LIN {X 0,Y 445.555,Z 224.747,A -85,B 0,C 180,E1 -8713.867,E2 -8713.867} C_VEL
LIN {X 0,Y 447.569,Z 235.644,A -85,B 0,C 180,E1 -8714.246,E2 -8714.246} C_VEL
LIN {X 0,Y 449.181,Z 245.497,A -85,B 0,C 180,E1 -8714.691,E2 -8714.691} C_VEL
LIN {X 0,Y 449.133,Z 253.576,A -85,B 0,C 180,E1 -8715.096,E2 -8715.096} C_VEL
LIN {X 0,Y 448.605,Z 263.719,A -85,B 0,C 180,E1 -8715.715,E2 -8715.715} C_VEL
LIN {X 0,Y 448.134,Z 272.72,A -85,B 0,C 180,E1 -8716.394,E2 -8716.394} C_VEL
LIN {X 0,Y 447.699,Z 281.135,A -85,B 0,C 180,E1 -8717.157,E2 -8717.157} C_VEL
LIN {X 0,Y 447.283,Z 288.853,A -85,B 0,C 180,E1 -8717.984,E2 -8717.984} C_VEL
LIN {X 0,Y 446.817,Z 296.075,A -85,B 0,C 180,E1 -8718.891,E2 -8718.891} C_VEL
LIN {X 0,Y 446.49,Z 302.281,A -85,B 0,C 180,E1 -8719.8,E2 -8719.8} C_VEL
LIN {X 0,Y 446.129,Z 308.821,A -85,B 0,C 180,E1 -8720.936,E2 -8720.936} C_VEL
LIN {X 0,Y 445.886,Z 313.324,A -85,B 0,C 180,E1 -8721.845,E2 -8721.845} C_VEL
LIN {X 0,Y 445.655,Z 318.973,A -85,B 0,C 180,E1 -8723.253,E2 -8723.253} C_VEL
LIN {X 0,Y 445.538,Z 323.142,A -85,B 0,C 180,E1 -8724.569,E2 -8724.569} C_VEL
LIN {X 0,Y 445.43,Z 325.507,A -85,B 0,C 180,E1 -8725.475,E2 -8725.475} C_VEL
LIN {X 0,Y 445.391,Z 327.304,A -85,B 0,C 180,E1 -8726.381,E2 -8726.381} C_VEL
LIN {X 0,Y 445.353,Z 329.747,A -85,B 0,C 180,E1 -8728.191,E2 -8728.191} C_VEL
LIN {X 0,Y 445.315,Z 330.334,A -85,B 0,C 180,E1 -8729.096,E2 -8729.096} C_VEL
LIN {X 0,Y 445.315,Z 330.334,A -85,B 0,C 180,E1 -8730.904,E2 -8730.904} C_VEL
LIN {X 0,Y 445.353,Z 329.747,A -85,B 0,C 180,E1 -8731.809,E2 -8731.809} C_VEL
LIN {X 0,Y 445.391,Z 327.304,A -85,B 0,C 180,E1 -8733.619,E2 -8733.619} C_VEL
LIN {X 0,Y 445.5,Z 324.359,A -85,B 0,C 180,E1 -8734.977,E2 -8734.977} C_VEL
LIN {X 0,Y 445.579,Z 320.37,A -85,B 0,C 180,E1 -8736.339,E2 -8736.339} C_VEL
LIN {X 0,Y 445.762,Z 315.239,A -85,B 0,C 180,E1 -8737.701,E2 -8737.701} C_VEL
LIN {X 0,Y 446.078,Z 309.978,A -85,B 0,C 180,E1 -8738.836,E2 -8738.836} C_VEL
LIN {X 0,Y 446.426,Z 303.658,A -85,B 0,C 180,E1 -8739.972,E2 -8739.972} C_VEL
LIN {X 0,Y 446.703,Z 297.702,A -85,B 0,C 180,E1 -8740.882,E2 -8740.882} C_VEL
LIN {X 0,Y 447.153,Z 290.773,A -85,B 0,C 180,E1 -8741.79,E2 -8741.79} C_VEL
LIN {X 0,Y 447.622,Z 282.589,A -85,B 0,C 180,E1 -8742.698,E2 -8742.698} C_VEL
LIN {X 0,Y 448.019,Z 274.012,A -85,B 0,C 180,E1 -8743.499,E2 -8743.499} C_VEL
LIN {X 0,Y 448.505,Z 265.351,A -85,B 0,C 180,E1 -8744.172,E2 -8744.172} C_VEL
LIN {X 0,Y 448.992,Z 255.589,A -85,B 0,C 180,E1 -8744.793,E2 -8744.793} C_VEL
LIN {X 0,Y 449.335,Z 246.791,A -85,B 0,C 180,E1 -8745.246,E2 -8745.246} C_VEL
LIN {X 0,Y 447.725,Z 236.462,A -85,B 0,C 180,E1 -8745.721,E2 -8745.721} C_VEL
LIN {X 0,Y 445.687,Z 225.777,A -85,B 0,C 180,E1 -8746.102,E2 -8746.102} C_VEL
LIN {X 0,Y 445.555,Z 224.693,A -85,B 0,C 180,E1 -8746.161,E2 -8746.161} C_VEL
LIN {X 0,Y 445.687,Z 218.655,A -85,B 0,C 180,E1 -8749.338,E2 -8749.338} C_VEL
LIN {X 0,Y 445.855,Z 213.313,A -85,B 0,C 180,E1 -8752.229,E2 -8752.229} C_VEL
LIN {X 0,Y 446.032,Z 208.032,A -85,B 0,C 180,E1 -8755.178,E2 -8755.178} C_VEL
LIN {X 0,Y 446.268,Z 202.816,A -85,B 0,C 180,E1 -8758.193,E2 -8758.193} C_VEL
LIN {X 0,Y 446.557,Z 196.849,A -85,B 0,C 180,E1 -8761.803,E2 -8761.803} C_VEL
LIN {X 0,Y 446.894,Z 191.658,A -85,B 0,C 180,E1 -8765.137,E2 -8765.137} C_VEL
LIN {X 0,Y 447.241,Z 187.135,A -85,B 0,C 180,E1 -8768.213,E2 -8768.213} C_VEL
LIN {X 0,Y 447.459,Z 182.971,A -85,B 0,C 180,E1 -8771.274,E2 -8771.274} C_VEL
LIN {X 0,Y 447.256,Z 179.884,A -85,B 0,C 180,E1 -8773.74,E2 -8773.74} C_VEL
LIN {X 0,Y 446.776,Z 176.867,A -85,B 0,C 180,E1 -8776.352,E2 -8776.352} C_VEL
LIN {X 0,Y 446.43,Z 174.429,A -85,B 0,C 180,E1 -8778.609,E2 -8778.609} C_VEL
LIN {X 0,Y 446.438,Z 174.378,A -85,B 0,C 180,E1 -8780.972,E2 -8780.972} C_VEL
LIN {X 0,Y 446.416,Z 174.377,A -85,B 0,C 180,E1 -8784.373,E2 -8784.373} C_VEL
LIN {X 0,Y 446.419,Z 174.373,A -85,B 0,C 180,E1 -8787.638,E2 -8787.638} C_VEL
LIN {X 0,Y 446.444,Z 174.374,A -85,B 0,C 180,E1 -8790.79,E2 -8790.79} C_VEL
LIN {X 0,Y 446.474,Z 174.367,A -85,B 0,C 180,E1 -8793.848,E2 -8793.848} C_VEL
LIN {X 0,Y 446.425,Z 174.375,A -85,B 0,C 180,E1 -8796.823,E2 -8796.823} C_VEL
LIN {X 0,Y 446.44,Z 174.372,A -85,B 0,C 180,E1 -8799.736,E2 -8799.736} C_VEL
LIN {X 0,Y 446.458,Z 174.371,A -85,B 0,C 180,E1 -8802.596,E2 -8802.596} C_VEL
LIN {X 0,Y 446.465,Z 174.368,A -85,B 0,C 180,E1 -8805.412,E2 -8805.412} C_VEL
LIN {X 0,Y 446.512,Z 174.367,A -85,B 0,C 180,E1 -8808.192,E2 -8808.192} C_VEL
LIN {X 0,Y 446.595,Z 174.358,A -85,B 0,C 180,E1 -8811.857,E2 -8811.857} C_VEL
LIN {X 0,Y 446.637,Z 174.346,A -85,B 0,C 180,E1 -8814.582,E2 -8814.582} C_VEL
LIN {X 0,Y 446.657,Z 174.346,A -85,B 0,C 180,E1 -8818.196,E2 -8818.196} C_VEL
LIN {X 0,Y 446.787,Z 174.331,A -85,B 0,C 180,E1 -8820,E2 -8820} C_VEL
LIN {X 0,Y 446.685,Z 174.34,A -85,B 0,C 180,E1 -8822.705,E2 -8822.705} C_VEL
LIN {X 0,Y 446.64,Z 174.346,A -85,B 0,C 180,E1 -8826.323,E2 -8826.323} C_VEL
LIN {X 0,Y 446.532,Z 174.362,A -85,B 0,C 180,E1 -8829.055,E2 -8829.055} C_VEL
LIN {X 0,Y 446.515,Z 174.362,A -85,B 0,C 180,E1 -8832.729,E2 -8832.729} C_VEL
LIN {X 0,Y 446.49,Z 174.364,A -85,B 0,C 180,E1 -8836.228,E2 -8836.228} C_VEL
LIN {X 0,Y 446.463,Z 174.373,A -85,B 0,C 180,E1 -8839.303,E2 -8839.303} C_VEL
LIN {X 0,Y 446.411,Z 174.374,A -85,B 0,C 180,E1 -8842.199,E2 -8842.199} C_VEL
LIN {X 0,Y 446.451,Z 174.374,A -85,B 0,C 180,E1 -8845.152,E2 -8845.152} C_VEL
LIN {X 0,Y 446.478,Z 174.366,A -85,B 0,C 180,E1 -8848.178,E2 -8848.178} C_VEL
LIN {X 0,Y 446.413,Z 174.375,A -85,B 0,C 180,E1 -8851.3,E2 -8851.3} C_VEL
LIN {X 0,Y 446.424,Z 174.378,A -85,B 0,C 180,E1 -8854.523,E2 -8854.523} C_VEL
LIN {X 0,Y 446.43,Z 174.374,A -85,B 0,C 180,E1 -8858.083,E2 -8858.083} C_VEL
LIN {X 0,Y 446.437,Z 174.373,A -85,B 0,C 180,E1 -8860.92,E2 -8860.92} C_VEL
LIN {X 0,Y 446.395,Z 174.378,A -85,B 0,C 180,E1 -8863.846,E2 -8863.846} C_VEL
LIN {X 0,Y 446.409,Z 174.381,A -85,B 0,C 180,E1 -8866.401,E2 -8866.401} C_VEL
LIN {X 0,Y 446.445,Z 174.373,A -85,B 0,C 180,E1 -8869.803,E2 -8869.803} C_VEL
LIN {X 0,Y 446.422,Z 174.38,A -85,B 0,C 180,E1 -8872.123,E2 -8872.123} C_VEL
LIN {X 0,Y 446.425,Z 174.374,A -85,B 0,C 180,E1 -8875.477,E2 -8875.477} C_VEL
LIN {X 0,Y 446.415,Z 174.374,A -85,B 0,C 180,E1 -8878.7,E2 -8878.7} C_VEL
LIN {X 0,Y 446.48,Z 174.373,A -85,B 0,C 180,E1 -8881.821,E2 -8881.821} C_VEL
LIN {X 0,Y 446.453,Z 174.369,A -85,B 0,C 180,E1 -8884.848,E2 -8884.848} C_VEL
LIN {X 0,Y 446.444,Z 174.371,A -85,B 0,C 180,E1 -8888.245,E2 -8888.245} C_VEL
LIN {X 0,Y 446.454,Z 174.376,A -85,B 0,C 180,E1 -8891.649,E2 -8891.649} C_VEL
LIN {X 0,Y 446.505,Z 174.366,A -85,B 0,C 180,E1 -8894.48,E2 -8894.48} C_VEL
LIN {X 0,Y 446.514,Z 174.364,A -85,B 0,C 180,E1 -8898.193,E2 -8898.193} C_VEL
LIN {X 0,Y 446.597,Z 174.355,A -85,B 0,C 180,E1 -8901.858,E2 -8901.858} C_VEL
LIN {X 0,Y 446.644,Z 174.349,A -85,B 0,C 180,E1 -8904.583,E2 -8904.583} C_VEL
LIN {X 0,Y 446.619,Z 174.353,A -85,B 0,C 180,E1 -8907.001,E2 -8907.001} C_VEL
LIN {X 0,Y 446.101,Z 174.421,A -85,B 0,C 180,E1 -8907.754,E2 -8907.754} C_VEL
LIN {X 0,Y 443.286,Z 174.777,A -85,B 0,C 180,E1 -8908.977,E2 -8908.977} C_VEL
LIN {X 0,Y 440.802,Z 175.085,A -85,B 0,C 180,E1 -8909.964,E2 -8909.964} C_VEL
LIN {X 0,Y 439.713,Z 175.216,A -85,B 0,C 180,E1 -8910.727,E2 -8910.727} C_VEL
LIN {X 0,Y 439.619,Z 175.225,A -85,B 0,C 180,E1 -8910.986,E2 -8910.986} C_VEL
LIN {X 0,Y 439.653,Z 175.222,A -85,B 0,C 180,E1 -8912.749,E2 -8912.749} C_VEL
LIN {X 0,Y 439.616,Z 175.227,A -85,B 0,C 180,E1 -8916.425,E2 -8916.425} C_VEL
LIN {X 0,Y 439.497,Z 175.24,A -85,B 0,C 180,E1 -8919.202,E2 -8919.202} C_VEL
LIN {X 0,Y 439.462,Z 175.246,A -85,B 0,C 180,E1 -8922.938,E2 -8922.938} C_VEL
LIN {X 0,Y 439.443,Z 175.248,A -85,B 0,C 180,E1 -8926.349,E2 -8926.349} C_VEL
LIN {X 0,Y 439.399,Z 175.248,A -85,B 0,C 180,E1 -8929.626,E2 -8929.626} C_VEL
LIN {X 0,Y 439.362,Z 175.256,A -85,B 0,C 180,E1 -8932.575,E2 -8932.575} C_VEL
LIN {X 0,Y 439.4,Z 175.248,A -85,B 0,C 180,E1 -8935.585,E2 -8935.585} C_VEL
LIN {X 0,Y 439.42,Z 175.246,A -85,B 0,C 180,E1 -8938.673,E2 -8938.673} C_VEL
LIN {X 0,Y 439.378,Z 175.258,A -85,B 0,C 180,E1 -8942.033,E2 -8942.033} C_VEL
LIN {X 0,Y 439.391,Z 175.25,A -85,B 0,C 180,E1 -8945.341,E2 -8945.341} C_VEL
LIN {X 0,Y 439.39,Z 175.249,A -85,B 0,C 180,E1 -8948.594,E2 -8948.594} C_VEL
LIN {X 0,Y 439.392,Z 175.25,A -85,B 0,C 180,E1 -8951.258,E2 -8951.258} C_VEL
LIN {X 0,Y 439.395,Z 175.248,A -85,B 0,C 180,E1 -8954.729,E2 -8954.729} C_VEL
LIN {X 0,Y 439.391,Z 175.253,A -85,B 0,C 180,E1 -8957.796,E2 -8957.796} C_VEL
LIN {X 0,Y 439.444,Z 175.242,A -85,B 0,C 180,E1 -8960.23,E2 -8960.23} C_VEL
LIN {X 0,Y 439.371,Z 175.255,A -85,B 0,C 180,E1 -8963.713,E2 -8963.713} C_VEL
LIN {X 0,Y 439.366,Z 175.256,A -85,B 0,C 180,E1 -8967.054,E2 -8967.054} C_VEL
LIN {X 0,Y 439.39,Z 175.249,A -85,B 0,C 180,E1 -8970.275,E2 -8970.275} C_VEL
LIN {X 0,Y 439.427,Z 175.246,A -85,B 0,C 180,E1 -8973.589,E2 -8973.589} C_VEL
LIN {X 0,Y 439.38,Z 175.251,A -85,B 0,C 180,E1 -8976.43,E2 -8976.43} C_VEL
LIN {X 0,Y 439.382,Z 175.252,A -85,B 0,C 180,E1 -8979.397,E2 -8979.397} C_VEL
LIN {X 0,Y 439.425,Z 175.246,A -85,B 0,C 180,E1 -8982.31,E2 -8982.31} C_VEL
LIN {X 0,Y 439.442,Z 175.245,A -85,B 0,C 180,E1 -8985.174,E2 -8985.174} C_VEL
LIN {X 0,Y 439.477,Z 175.239,A -85,B 0,C 180,E1 -8988.002,E2 -8988.002} C_VEL
LIN {X 0,Y 439.542,Z 175.23,A -85,B 0,C 180,E1 -8991.727,E2 -8991.727} C_VEL
LIN {X 0,Y 439.614,Z 175.228,A -85,B 0,C 180,E1 -8994.496,E2 -8994.496} C_VEL
LIN {X 0,Y 439.628,Z 175.224,A -85,B 0,C 180,E1 -8998.168,E2 -8998.168} C_VEL
LIN {X 0,Y 439.757,Z 175.206,A -85,B 0,C 180,E1 -9000,E2 -9000} C_VEL
LIN {X 0,Y 439.634,Z 175.22,A -85,B 0,C 180,E1 -9002.749,E2 -9002.749} C_VEL
LIN {X 0,Y 439.607,Z 175.225,A -85,B 0,C 180,E1 -9006.426,E2 -9006.426} C_VEL
LIN {X 0,Y 439.495,Z 175.236,A -85,B 0,C 180,E1 -9009.202,E2 -9009.202} C_VEL
LIN {X 0,Y 439.461,Z 175.24,A -85,B 0,C 180,E1 -9012.938,E2 -9012.938} C_VEL
LIN {X 0,Y 439.443,Z 175.244,A -85,B 0,C 180,E1 -9016.349,E2 -9016.349} C_VEL
LIN {X 0,Y 439.398,Z 175.254,A -85,B 0,C 180,E1 -9019.627,E2 -9019.627} C_VEL
LIN {X 0,Y 439.361,Z 175.252,A -85,B 0,C 180,E1 -9022.576,E2 -9022.576} C_VEL
LIN {X 0,Y 439.402,Z 175.254,A -85,B 0,C 180,E1 -9025.586,E2 -9025.586} C_VEL
LIN {X 0,Y 439.414,Z 175.246,A -85,B 0,C 180,E1 -9028.674,E2 -9028.674} C_VEL
LIN {X 0,Y 439.367,Z 175.252,A -85,B 0,C 180,E1 -9032.031,E2 -9032.031} C_VEL
LIN {X 0,Y 439.392,Z 175.255,A -85,B 0,C 180,E1 -9035.341,E2 -9035.341} C_VEL
LIN {X 0,Y 439.375,Z 175.257,A -85,B 0,C 180,E1 -9038.596,E2 -9038.596} C_VEL
LIN {X 0,Y 439.378,Z 175.258,A -85,B 0,C 180,E1 -9040.982,E2 -9040.982} C_VEL
LIN {X 0,Y 439.858,Z 178.467,A -85,B 0,C 180,E1 -9044.029,E2 -9044.029} C_VEL
LIN {X 0,Y 440.283,Z 181.496,A -85,B 0,C 180,E1 -9046.656,E2 -9046.656} C_VEL
LIN {X 0,Y 440.452,Z 184.61,A -85,B 0,C 180,E1 -9049.141,E2 -9049.141} C_VEL
LIN {X 0,Y 440.242,Z 187.779,A -85,B 0,C 180,E1 -9051.495,E2 -9051.495} C_VEL
LIN {X 0,Y 439.847,Z 192.663,A -85,B 0,C 180,E1 -9054.886,E2 -9054.886} C_VEL
LIN {X 0,Y 439.507,Z 197.659,A -85,B 0,C 180,E1 -9058.151,E2 -9058.151} C_VEL
LIN {X 0,Y 439.237,Z 202.762,A -85,B 0,C 180,E1 -9061.314,E2 -9061.314} C_VEL
LIN {X 0,Y 438.997,Z 207.948,A -85,B 0,C 180,E1 -9064.39,E2 -9064.39} C_VEL
LIN {X 0,Y 438.785,Z 213.194,A -85,B 0,C 180,E1 -9067.393,E2 -9067.393} C_VEL
LIN {X 0,Y 438.613,Z 218.502,A -85,B 0,C 180,E1 -9070.337,E2 -9070.337} C_VEL
LIN {X 0,Y 438.483,Z 224.562,A -85,B 0,C 180,E1 -9073.599,E2 -9073.599} C_VEL
LIN {X 0,Y 440.39,Z 234.647,A -85,B 0,C 180,E1 -9073.956,E2 -9073.956} C_VEL
LIN {X 0,Y 441.936,Z 243.984,A -85,B 0,C 180,E1 -9074.374,E2 -9074.374} C_VEL
LIN {X 0,Y 442.45,Z 249.156,A -85,B 0,C 180,E1 -9074.629,E2 -9074.629} C_VEL
LIN {X 0,Y 441.776,Z 261.874,A -85,B 0,C 180,E1 -9075.372,E2 -9075.372} C_VEL
LIN {X 0,Y 441.28,Z 271.155,A -85,B 0,C 180,E1 -9076.061,E2 -9076.061} C_VEL
LIN {X 0,Y 440.804,Z 279.838,A -85,B 0,C 180,E1 -9076.841,E2 -9076.841} C_VEL
LIN {X 0,Y 440.318,Z 288.641,A -85,B 0,C 180,E1 -9077.791,E2 -9077.791} C_VEL
LIN {X 0,Y 439.825,Z 295.863,A -85,B 0,C 180,E1 -9078.712,E2 -9078.712} C_VEL
LIN {X 0,Y 439.469,Z 302.069,A -85,B 0,C 180,E1 -9079.636,E2 -9079.636} C_VEL
LIN {X 0,Y 439.085,Z 308.609,A -85,B 0,C 180,E1 -9080.79,E2 -9080.79} C_VEL
LIN {X 0,Y 438.832,Z 313.112,A -85,B 0,C 180,E1 -9081.713,E2 -9081.713} C_VEL
LIN {X 0,Y 438.591,Z 318.605,A -85,B 0,C 180,E1 -9083.098,E2 -9083.098} C_VEL
LIN {X 0,Y 438.438,Z 322.93,A -85,B 0,C 180,E1 -9084.481,E2 -9084.481} C_VEL
LIN {X 0,Y 438.36,Z 325.296,A -85,B 0,C 180,E1 -9085.402,E2 -9085.402} C_VEL
LIN {X 0,Y 438.333,Z 328.481,A -85,B 0,C 180,E1 -9087.243,E2 -9087.243} C_VEL
LIN {X 0,Y 438.275,Z 329.536,A -85,B 0,C 180,E1 -9088.162,E2 -9088.162} C_VEL
LIN {X 0,Y 438.23,Z 330.123,A -85,B 0,C 180,E1 -9089.081,E2 -9089.081} C_VEL
LIN {X 0,Y 438.23,Z 330.123,A -85,B 0,C 180,E1 -9090.919,E2 -9090.919} C_VEL
LIN {X 0,Y 438.275,Z 329.536,A -85,B 0,C 180,E1 -9091.838,E2 -9091.838} C_VEL
LIN {X 0,Y 438.292,Z 327.093,A -85,B 0,C 180,E1 -9093.677,E2 -9093.677} C_VEL
LIN {X 0,Y 438.414,Z 324.147,A -85,B 0,C 180,E1 -9095.058,E2 -9095.058} C_VEL
LIN {X 0,Y 438.507,Z 320.158,A -85,B 0,C 180,E1 -9096.441,E2 -9096.441} C_VEL
LIN {X 0,Y 438.718,Z 315.028,A -85,B 0,C 180,E1 -9097.826,E2 -9097.826} C_VEL
LIN {X 0,Y 439.038,Z 309.765,A -85,B 0,C 180,E1 -9098.979,E2 -9098.979} C_VEL
LIN {X 0,Y 439.397,Z 303.446,A -85,B 0,C 180,E1 -9100.133,E2 -9100.133} C_VEL
LIN {X 0,Y 439.697,Z 297.49,A -85,B 0,C 180,E1 -9101.058,E2 -9101.058} C_VEL
LIN {X 0,Y 440.192,Z 290.561,A -85,B 0,C 180,E1 -9101.979,E2 -9101.979} C_VEL
LIN {X 0,Y 440.663,Z 282.377,A -85,B 0,C 180,E1 -9102.902,E2 -9102.902} C_VEL
LIN {X 0,Y 441.074,Z 274.078,A -85,B 0,C 180,E1 -9103.691,E2 -9103.691} C_VEL
LIN {X 0,Y 441.592,Z 265.139,A -85,B 0,C 180,E1 -9104.399,E2 -9104.399} C_VEL
LIN {X 0,Y 442.134,Z 255.378,A -85,B 0,C 180,E1 -9105.028,E2 -9105.028} C_VEL
LIN {X 0,Y 442.464,Z 247.869,A -85,B 0,C 180,E1 -9105.429,E2 -9105.429} C_VEL
LIN {X 0,Y 440.705,Z 236.497,A -85,B 0,C 180,E1 -9105.97,E2 -9105.97} C_VEL
LIN {X 0,Y 438.589,Z 225.608,A -85,B 0,C 180,E1 -9106.368,E2 -9106.368} C_VEL
LIN {X 0,Y 438.483,Z 224.562,A -85,B 0,C 180,E1 -9106.401,E2 -9106.401} C_VEL
LIN {X 0,Y 438.611,Z 218.499,A -85,B 0,C 180,E1 -9109.663,E2 -9109.663} C_VEL
LIN {X 0,Y 438.785,Z 213.188,A -85,B 0,C 180,E1 -9112.607,E2 -9112.607} C_VEL
LIN {X 0,Y 438.997,Z 207.939,A -85,B 0,C 180,E1 -9115.61,E2 -9115.61} C_VEL
LIN {X 0,Y 439.236,Z 202.751,A -85,B 0,C 180,E1 -9118.686,E2 -9118.686} C_VEL
LIN {X 0,Y 439.527,Z 197.323,A -85,B 0,C 180,E1 -9122.062,E2 -9122.062} C_VEL
LIN {X 0,Y 439.849,Z 192.655,A -85,B 0,C 180,E1 -9125.114,E2 -9125.114} C_VEL
LIN {X 0,Y 440.245,Z 187.739,A -85,B 0,C 180,E1 -9128.534,E2 -9128.534} C_VEL
LIN {X 0,Y 440.437,Z 183.892,A -85,B 0,C 180,E1 -9131.411,E2 -9131.411} C_VEL
LIN {X 0,Y 440.198,Z 180.623,A -85,B 0,C 180,E1 -9134.073,E2 -9134.073} C_VEL
LIN {X 0,Y 439.643,Z 177.006,A -85,B 0,C 180,E1 -9137.335,E2 -9137.335} C_VEL
LIN {X 0,Y 439.378,Z 175.257,A -85,B 0,C 180,E1 -9139.018,E2 -9139.018} C_VEL
LIN {X 0,Y 439.371,Z 175.256,A -85,B 0,C 180,E1 -9141.607,E2 -9141.607} C_VEL
LIN {X 0,Y 439.396,Z 175.255,A -85,B 0,C 180,E1 -9144.843,E2 -9144.843} C_VEL
LIN {X 0,Y 439.37,Z 175.253,A -85,B 0,C 180,E1 -9148.139,E2 -9148.139} C_VEL
LIN {X 0,Y 439.429,Z 175.244,A -85,B 0,C 180,E1 -9151.597,E2 -9151.597} C_VEL
LIN {X 0,Y 439.402,Z 175.254,A -85,B 0,C 180,E1 -9154.414,E2 -9154.414} C_VEL
LIN {X 0,Y 439.361,Z 175.252,A -85,B 0,C 180,E1 -9157.424,E2 -9157.424} C_VEL
LIN {X 0,Y 439.437,Z 175.245,A -85,B 0,C 180,E1 -9160.662,E2 -9160.662} C_VEL
LIN {X 0,Y 439.458,Z 175.247,A -85,B 0,C 180,E1 -9164.224,E2 -9164.224} C_VEL
LIN {X 0,Y 439.479,Z 175.245,A -85,B 0,C 180,E1 -9168.001,E2 -9168.001} C_VEL
LIN {X 0,Y 439.543,Z 175.234,A -85,B 0,C 180,E1 -9171.726,E2 -9171.726} C_VEL
LIN {X 0,Y 439.612,Z 175.222,A -85,B 0,C 180,E1 -9174.495,E2 -9174.495} C_VEL
LIN {X 0,Y 439.627,Z 175.222,A -85,B 0,C 180,E1 -9178.167,E2 -9178.167} C_VEL
LIN {X 0,Y 439.757,Z 175.206,A -85,B 0,C 180,E1 -9180,E2 -9180} C_VEL
LIN {X 0,Y 439.635,Z 175.218,A -85,B 0,C 180,E1 -9182.748,E2 -9182.748} C_VEL
LIN {X 0,Y 439.611,Z 175.221,A -85,B 0,C 180,E1 -9186.425,E2 -9186.425} C_VEL
LIN {X 0,Y 439.494,Z 175.24,A -85,B 0,C 180,E1 -9189.201,E2 -9189.201} C_VEL
LIN {X 0,Y 439.459,Z 175.243,A -85,B 0,C 180,E1 -9192.937,E2 -9192.937} C_VEL
LIN {X 0,Y 439.441,Z 175.242,A -85,B 0,C 180,E1 -9196.348,E2 -9196.348} C_VEL
LIN {X 0,Y 439.396,Z 175.249,A -85,B 0,C 180,E1 -9199.626,E2 -9199.626} C_VEL
LIN {X 0,Y 439.358,Z 175.255,A -85,B 0,C 180,E1 -9202.575,E2 -9202.575} C_VEL
LIN {X 0,Y 439.398,Z 175.248,A -85,B 0,C 180,E1 -9205.585,E2 -9205.585} C_VEL
LIN {X 0,Y 439.419,Z 175.25,A -85,B 0,C 180,E1 -9208.673,E2 -9208.673} C_VEL
LIN {X 0,Y 439.367,Z 175.251,A -85,B 0,C 180,E1 -9211.86,E2 -9211.86} C_VEL
LIN {X 0,Y 439.394,Z 175.25,A -85,B 0,C 180,E1 -9215.156,E2 -9215.156} C_VEL
LIN {X 0,Y 439.391,Z 175.255,A -85,B 0,C 180,E1 -9218.593,E2 -9218.593} C_VEL
LIN {X 0,Y 439.392,Z 175.249,A -85,B 0,C 180,E1 -9221.258,E2 -9221.258} C_VEL
LIN {X 0,Y 439.395,Z 175.251,A -85,B 0,C 180,E1 -9224.729,E2 -9224.729} C_VEL
LIN {X 0,Y 439.39,Z 175.251,A -85,B 0,C 180,E1 -9227.796,E2 -9227.796} C_VEL
LIN {X 0,Y 439.431,Z 175.251,A -85,B 0,C 180,E1 -9230.229,E2 -9230.229} C_VEL
LIN {X 0,Y 439.372,Z 175.254,A -85,B 0,C 180,E1 -9233.713,E2 -9233.713} C_VEL
LIN {X 0,Y 439.37,Z 175.251,A -85,B 0,C 180,E1 -9237.054,E2 -9237.054} C_VEL
LIN {X 0,Y 439.392,Z 175.251,A -85,B 0,C 180,E1 -9240.275,E2 -9240.275} C_VEL
LIN {X 0,Y 439.429,Z 175.249,A -85,B 0,C 180,E1 -9243.589,E2 -9243.589} C_VEL
LIN {X 0,Y 439.383,Z 175.25,A -85,B 0,C 180,E1 -9246.43,E2 -9246.43} C_VEL
LIN {X 0,Y 439.385,Z 175.254,A -85,B 0,C 180,E1 -9249.397,E2 -9249.397} C_VEL
LIN {X 0,Y 439.428,Z 175.248,A -85,B 0,C 180,E1 -9252.31,E2 -9252.31} C_VEL
LIN {X 0,Y 439.446,Z 175.248,A -85,B 0,C 180,E1 -9255.174,E2 -9255.174} C_VEL
LIN {X 0,Y 439.48,Z 175.24,A -85,B 0,C 180,E1 -9258.001,E2 -9258.001} C_VEL
LIN {X 0,Y 439.544,Z 175.234,A -85,B 0,C 180,E1 -9261.726,E2 -9261.726} C_VEL
LIN {X 0,Y 439.619,Z 175.224,A -85,B 0,C 180,E1 -9264.496,E2 -9264.496} C_VEL
LIN {X 0,Y 439.633,Z 175.221,A -85,B 0,C 180,E1 -9268.168,E2 -9268.168} C_VEL
LIN {X 0,Y 439.761,Z 175.207,A -85,B 0,C 180,E1 -9270,E2 -9270} C_VEL
LIN {X 0,Y 439.619,Z 175.225,A -85,B 0,C 180,E1 -9270.986,E2 -9270.986} C_VEL
LIN {X 0,Y 438.902,Z 175.313,A -85,B 0,C 180,E1 -9271.75,E2 -9271.75} C_VEL
LIN {X 0,Y 435.924,Z 175.686,A -85,B 0,C 180,E1 -9272.989,E2 -9272.989} C_VEL
LIN {X 0,Y 433.472,Z 175.992,A -85,B 0,C 180,E1 -9273.989,E2 -9273.989} C_VEL
LIN {X 0,Y 432.499,Z 176.113,A -85,B 0,C 180,E1 -9274.764,E2 -9274.764} C_VEL
LIN {X 0,Y 432.462,Z 176.115,A -85,B 0,C 180,E1 -9275.026,E2 -9275.026} C_VEL
LIN {X 0,Y 432.582,Z 176.101,A -85,B 0,C 180,E1 -9277.679,E2 -9277.679} C_VEL
LIN {X 0,Y 432.389,Z 176.125,A -85,B 0,C 180,E1 -9281.247,E2 -9281.247} C_VEL
LIN {X 0,Y 432.371,Z 176.128,A -85,B 0,C 180,E1 -9284.112,E2 -9284.112} C_VEL
LIN {X 0,Y 432.393,Z 176.126,A -85,B 0,C 180,E1 -9287.011,E2 -9287.011} C_VEL
LIN {X 0,Y 432.335,Z 176.13,A -85,B 0,C 180,E1 -9289.96,E2 -9289.96} C_VEL
LIN {X 0,Y 432.315,Z 176.131,A -85,B 0,C 180,E1 -9292.964,E2 -9292.964} C_VEL
LIN {X 0,Y 432.36,Z 176.129,A -85,B 0,C 180,E1 -9296.032,E2 -9296.032} C_VEL
LIN {X 0,Y 432.348,Z 176.126,A -85,B 0,C 180,E1 -9299.187,E2 -9299.187} C_VEL
LIN {X 0,Y 432.327,Z 176.133,A -85,B 0,C 180,E1 -9302.295,E2 -9302.295} C_VEL
LIN {X 0,Y 432.336,Z 176.128,A -85,B 0,C 180,E1 -9304.677,E2 -9304.677} C_VEL
LIN {X 0,Y 432.345,Z 176.13,A -85,B 0,C 180,E1 -9308.148,E2 -9308.148} C_VEL
LIN {X 0,Y 432.361,Z 176.13,A -85,B 0,C 180,E1 -9311.607,E2 -9311.607} C_VEL
LIN {X 0,Y 432.327,Z 176.129,A -85,B 0,C 180,E1 -9314.347,E2 -9314.347} C_VEL
LIN {X 0,Y 432.314,Z 176.131,A -85,B 0,C 180,E1 -9317.016,E2 -9317.016} C_VEL
LIN {X 0,Y 432.35,Z 176.129,A -85,B 0,C 180,E1 -9319.817,E2 -9319.817} C_VEL
LIN {X 0,Y 432.31,Z 176.133,A -85,B 0,C 180,E1 -9323.023,E2 -9323.023} C_VEL
LIN {X 0,Y 432.353,Z 176.126,A -85,B 0,C 180,E1 -9325.997,E2 -9325.997} C_VEL
LIN {X 0,Y 432.388,Z 176.122,A -85,B 0,C 180,E1 -9329.744,E2 -9329.744} C_VEL
LIN {X 0,Y 432.393,Z 176.124,A -85,B 0,C 180,E1 -9333.373,E2 -9333.373} C_VEL
LIN {X 0,Y 432.365,Z 176.124,A -85,B 0,C 180,E1 -9336.024,E2 -9336.024} C_VEL
LIN {X 0,Y 432.344,Z 176.132,A -85,B 0,C 180,E1 -9339.046,E2 -9339.046} C_VEL
LIN {X 0,Y 432.371,Z 176.123,A -85,B 0,C 180,E1 -9342.011,E2 -9342.011} C_VEL
LIN {X 0,Y 432.39,Z 176.126,A -85,B 0,C 180,E1 -9344.927,E2 -9344.927} C_VEL
LIN {X 0,Y 432.453,Z 176.113,A -85,B 0,C 180,E1 -9347.804,E2 -9347.804} C_VEL
LIN {X 0,Y 432.486,Z 176.109,A -85,B 0,C 180,E1 -9351.591,E2 -9351.591} C_VEL
LIN {X 0,Y 432.591,Z 176.102,A -85,B 0,C 180,E1 -9354.407,E2 -9354.407} C_VEL
LIN {X 0,Y 432.598,Z 176.099,A -85,B 0,C 180,E1 -9358.139,E2 -9358.139} C_VEL
LIN {X 0,Y 432.727,Z 176.082,A -85,B 0,C 180,E1 -9360.001,E2 -9360.001} C_VEL
LIN {X 0,Y 432.586,Z 176.098,A -85,B 0,C 180,E1 -9362.794,E2 -9362.794} C_VEL
LIN {X 0,Y 432.56,Z 176.102,A -85,B 0,C 180,E1 -9366.531,E2 -9366.531} C_VEL
LIN {X 0,Y 432.438,Z 176.115,A -85,B 0,C 180,E1 -9369.354,E2 -9369.354} C_VEL
LIN {X 0,Y 432.426,Z 176.116,A -85,B 0,C 180,E1 -9372.804,E2 -9372.804} C_VEL
LIN {X 0,Y 432.408,Z 176.119,A -85,B 0,C 180,E1 -9376.479,E2 -9376.479} C_VEL
LIN {X 0,Y 432.334,Z 176.132,A -85,B 0,C 180,E1 -9379.961,E2 -9379.961} C_VEL
LIN {X 0,Y 432.316,Z 176.131,A -85,B 0,C 180,E1 -9382.965,E2 -9382.965} C_VEL
LIN {X 0,Y 432.361,Z 176.126,A -85,B 0,C 180,E1 -9386.033,E2 -9386.033} C_VEL
LIN {X 0,Y 432.339,Z 176.131,A -85,B 0,C 180,E1 -9389.188,E2 -9389.188} C_VEL
LIN {X 0,Y 432.32,Z 176.129,A -85,B 0,C 180,E1 -9392.444,E2 -9392.444} C_VEL
LIN {X 0,Y 432.341,Z 176.132,A -85,B 0,C 180,E1 -9395.633,E2 -9395.633} C_VEL
LIN {X 0,Y 432.337,Z 176.134,A -85,B 0,C 180,E1 -9398.715,E2 -9398.715} C_VEL
LIN {X 0,Y 432.321,Z 176.135,A -85,B 0,C 180,E1 -9400.562,E2 -9400.562} C_VEL
LIN {X 0,Y 432.727,Z 178.574,A -85,B 0,C 180,E1 -9403.043,E2 -9403.043} C_VEL
LIN {X 0,Y 433.174,Z 181.587,A -85,B 0,C 180,E1 -9405.762,E2 -9405.762} C_VEL
LIN {X 0,Y 433.427,Z 184.674,A -85,B 0,C 180,E1 -9408.333,E2 -9408.333} C_VEL
LIN {X 0,Y 433.277,Z 187.811,A -85,B 0,C 180,E1 -9410.758,E2 -9410.758} C_VEL
LIN {X 0,Y 432.872,Z 192.713,A -85,B 0,C 180,E1 -9414.272,E2 -9414.272} C_VEL
LIN {X 0,Y 432.503,Z 197.777,A -85,B 0,C 180,E1 -9417.67,E2 -9417.67} C_VEL
LIN {X 0,Y 432.212,Z 202.694,A -85,B 0,C 180,E1 -9420.803,E2 -9420.803} C_VEL
LIN {X 0,Y 431.978,Z 207.85,A -85,B 0,C 180,E1 -9423.943,E2 -9423.943} C_VEL
LIN {X 0,Y 431.731,Z 213.073,A -85,B 0,C 180,E1 -9427.003,E2 -9427.003} C_VEL
LIN {X 0,Y 431.539,Z 218.345,A -85,B 0,C 180,E1 -9430.001,E2 -9430.001} C_VEL
LIN {X 0,Y 431.4,Z 224.389,A -85,B 0,C 180,E1 -9433.328,E2 -9433.328} C_VEL
LIN {X 0,Y 433.3,Z 234.391,A -85,B 0,C 180,E1 -9433.685,E2 -9433.685} C_VEL
LIN {X 0,Y 434.878,Z 243.765,A -85,B 0,C 180,E1 -9434.114,E2 -9434.114} C_VEL
LIN {X 0,Y 435.537,Z 250.109,A -85,B 0,C 180,E1 -9434.439,E2 -9434.439} C_VEL
LIN {X 0,Y 434.893,Z 261.662,A -85,B 0,C 180,E1 -9435.135,E2 -9435.135} C_VEL
LIN {X 0,Y 434.364,Z 270.943,A -85,B 0,C 180,E1 -9435.835,E2 -9435.835} C_VEL
LIN {X 0,Y 433.818,Z 280.406,A -85,B 0,C 180,E1 -9436.707,E2 -9436.707} C_VEL
LIN {X 0,Y 433.367,Z 288.43,A -85,B 0,C 180,E1 -9437.592,E2 -9437.592} C_VEL
LIN {X 0,Y 432.845,Z 295.651,A -85,B 0,C 180,E1 -9438.528,E2 -9438.528} C_VEL
LIN {X 0,Y 432.456,Z 301.856,A -85,B 0,C 180,E1 -9439.466,E2 -9439.466} C_VEL
LIN {X 0,Y 432.059,Z 308.397,A -85,B 0,C 180,E1 -9440.639,E2 -9440.639} C_VEL
LIN {X 0,Y 431.79,Z 312.9,A -85,B 0,C 180,E1 -9441.577,E2 -9441.577} C_VEL
LIN {X 0,Y 431.521,Z 318.393,A -85,B 0,C 180,E1 -9442.984,E2 -9442.984} C_VEL
LIN {X 0,Y 431.343,Z 322.718,A -85,B 0,C 180,E1 -9444.39,E2 -9444.39} C_VEL
LIN {X 0,Y 431.29,Z 325.085,A -85,B 0,C 180,E1 -9445.327,E2 -9445.327} C_VEL
LIN {X 0,Y 431.23,Z 328.269,A -85,B 0,C 180,E1 -9447.198,E2 -9447.198} C_VEL
LIN {X 0,Y 431.2,Z 329.326,A -85,B 0,C 180,E1 -9448.132,E2 -9448.132} C_VEL
LIN {X 0,Y 431.149,Z 329.912,A -85,B 0,C 180,E1 -9449.066,E2 -9449.066} C_VEL
LIN {X 0,Y 431.149,Z 329.912,A -85,B 0,C 180,E1 -9450.934,E2 -9450.934} C_VEL
LIN {X 0,Y 431.2,Z 329.326,A -85,B 0,C 180,E1 -9451.868,E2 -9451.868} C_VEL
LIN {X 0,Y 431.199,Z 326.881,A -85,B 0,C 180,E1 -9453.738,E2 -9453.738} C_VEL
LIN {X 0,Y 431.329,Z 323.935,A -85,B 0,C 180,E1 -9455.141,E2 -9455.141} C_VEL
LIN {X 0,Y 431.442,Z 319.947,A -85,B 0,C 180,E1 -9456.547,E2 -9456.547} C_VEL
LIN {X 0,Y 431.646,Z 314.815,A -85,B 0,C 180,E1 -9457.955,E2 -9457.955} C_VEL
LIN {X 0,Y 431.973,Z 309.553,A -85,B 0,C 180,E1 -9459.127,E2 -9459.127} C_VEL
LIN {X 0,Y 432.357,Z 303.233,A -85,B 0,C 180,E1 -9460.3,E2 -9460.3} C_VEL
LIN {X 0,Y 432.704,Z 297.278,A -85,B 0,C 180,E1 -9461.239,E2 -9461.239} C_VEL
LIN {X 0,Y 433.226,Z 290.349,A -85,B 0,C 180,E1 -9462.174,E2 -9462.174} C_VEL
LIN {X 0,Y 433.726,Z 282.165,A -85,B 0,C 180,E1 -9463.112,E2 -9463.112} C_VEL
LIN {X 0,Y 434.188,Z 273.295,A -85,B 0,C 180,E1 -9463.963,E2 -9463.963} C_VEL
LIN {X 0,Y 434.717,Z 264.928,A -85,B 0,C 180,E1 -9464.632,E2 -9464.632} C_VEL
LIN {X 0,Y 435.279,Z 255.167,A -85,B 0,C 180,E1 -9465.271,E2 -9465.271} C_VEL
LIN {X 0,Y 435.429,Z 247.652,A -85,B 0,C 180,E1 -9465.685,E2 -9465.685} C_VEL
LIN {X 0,Y 433.582,Z 236.045,A -85,B 0,C 180,E1 -9466.248,E2 -9466.248} C_VEL
LIN {X 0,Y 431.512,Z 225.399,A -85,B 0,C 180,E1 -9466.644,E2 -9466.644} C_VEL
LIN {X 0,Y 431.396,Z 224.354,A -85,B 0,C 180,E1 -9466.691,E2 -9466.691} C_VEL
LIN {X 0,Y 431.536,Z 218.343,A -85,B 0,C 180,E1 -9469.999,E2 -9469.999} C_VEL
LIN {X 0,Y 431.731,Z 213.067,A -85,B 0,C 180,E1 -9472.997,E2 -9472.997} C_VEL
LIN {X 0,Y 432.015,Z 207.051,A -85,B 0,C 180,E1 -9476.524,E2 -9476.524} C_VEL
LIN {X 0,Y 432.202,Z 202.686,A -85,B 0,C 180,E1 -9479.197,E2 -9479.197} C_VEL
LIN {X 0,Y 432.511,Z 197.623,A -85,B 0,C 180,E1 -9482.427,E2 -9482.427} C_VEL
LIN {X 0,Y 432.875,Z 192.655,A -85,B 0,C 180,E1 -9485.766,E2 -9485.766} C_VEL
LIN {X 0,Y 433.241,Z 188.325,A -85,B 0,C 180,E1 -9488.862,E2 -9488.862} C_VEL
LIN {X 0,Y 433.41,Z 184.673,A -85,B 0,C 180,E1 -9491.669,E2 -9491.669} C_VEL
LIN {X 0,Y 433.148,Z 181.351,A -85,B 0,C 180,E1 -9494.445,E2 -9494.445} C_VEL
LIN {X 0,Y 432.7,Z 178.55,A -85,B 0,C 180,E1 -9496.986,E2 -9496.986} C_VEL
LIN {X 0,Y 432.321,Z 176.135,A -85,B 0,C 180,E1 -9499.438,E2 -9499.438} C_VEL
LIN {X 0,Y 432.334,Z 176.133,A -85,B 0,C 180,E1 -9501.849,E2 -9501.849} C_VEL
LIN {X 0,Y 432.337,Z 176.132,A -85,B 0,C 180,E1 -9505.322,E2 -9505.322} C_VEL
LIN {X 0,Y 432.318,Z 176.137,A -85,B 0,C 180,E1 -9508.653,E2 -9508.653} C_VEL
LIN {X 0,Y 432.378,Z 176.123,A -85,B 0,C 180,E1 -9511.876,E2 -9511.876} C_VEL
LIN {X 0,Y 432.348,Z 176.127,A -85,B 0,C 180,E1 -9514.998,E2 -9514.998} C_VEL
LIN {X 0,Y 432.354,Z 176.129,A -85,B 0,C 180,E1 -9518.045,E2 -9518.045} C_VEL
LIN {X 0,Y 432.382,Z 176.122,A -85,B 0,C 180,E1 -9521.029,E2 -9521.029} C_VEL
LIN {X 0,Y 432.426,Z 176.121,A -85,B 0,C 180,E1 -9523.96,E2 -9523.96} C_VEL
LIN {X 0,Y 432.454,Z 176.117,A -85,B 0,C 180,E1 -9527.803,E2 -9527.803} C_VEL
LIN {X 0,Y 432.487,Z 176.112,A -85,B 0,C 180,E1 -9531.59,E2 -9531.59} C_VEL
LIN {X 0,Y 432.589,Z 176.097,A -85,B 0,C 180,E1 -9534.406,E2 -9534.406} C_VEL
LIN {X 0,Y 432.597,Z 176.098,A -85,B 0,C 180,E1 -9538.138,E2 -9538.138} C_VEL
LIN {X 0,Y 432.727,Z 176.082,A -85,B 0,C 180,E1 -9539.999,E2 -9539.999} C_VEL
LIN {X 0,Y 432.586,Z 176.096,A -85,B 0,C 180,E1 -9542.793,E2 -9542.793} C_VEL
LIN {X 0,Y 432.566,Z 176.099,A -85,B 0,C 180,E1 -9546.53,E2 -9546.53} C_VEL
LIN {X 0,Y 432.436,Z 176.122,A -85,B 0,C 180,E1 -9549.353,E2 -9549.353} C_VEL
LIN {X 0,Y 432.425,Z 176.118,A -85,B 0,C 180,E1 -9552.803,E2 -9552.803} C_VEL
LIN {X 0,Y 432.406,Z 176.119,A -85,B 0,C 180,E1 -9556.479,E2 -9556.479} C_VEL
LIN {X 0,Y 432.332,Z 176.128,A -85,B 0,C 180,E1 -9559.96,E2 -9559.96} C_VEL
LIN {X 0,Y 432.312,Z 176.137,A -85,B 0,C 180,E1 -9562.964,E2 -9562.964} C_VEL
LIN {X 0,Y 432.358,Z 176.125,A -85,B 0,C 180,E1 -9566.032,E2 -9566.032} C_VEL
LIN {X 0,Y 432.346,Z 176.129,A -85,B 0,C 180,E1 -9569.187,E2 -9569.187} C_VEL
LIN {X 0,Y 432.319,Z 176.132,A -85,B 0,C 180,E1 -9572.293,E2 -9572.293} C_VEL
LIN {X 0,Y 432.334,Z 176.135,A -85,B 0,C 180,E1 -9574.677,E2 -9574.677} C_VEL
LIN {X 0,Y 432.346,Z 176.129,A -85,B 0,C 180,E1 -9578.148,E2 -9578.148} C_VEL
LIN {X 0,Y 432.36,Z 176.124,A -85,B 0,C 180,E1 -9581.607,E2 -9581.607} C_VEL
LIN {X 0,Y 432.327,Z 176.136,A -85,B 0,C 180,E1 -9584.347,E2 -9584.347} C_VEL
LIN {X 0,Y 432.317,Z 176.13,A -85,B 0,C 180,E1 -9587.015,E2 -9587.015} C_VEL
LIN {X 0,Y 432.335,Z 176.13,A -85,B 0,C 180,E1 -9589.82,E2 -9589.82} C_VEL
LIN {X 0,Y 432.31,Z 176.131,A -85,B 0,C 180,E1 -9593.023,E2 -9593.023} C_VEL
LIN {X 0,Y 432.354,Z 176.132,A -85,B 0,C 180,E1 -9595.997,E2 -9595.997} C_VEL
LIN {X 0,Y 432.39,Z 176.126,A -85,B 0,C 180,E1 -9599.744,E2 -9599.744} C_VEL
LIN {X 0,Y 432.395,Z 176.122,A -85,B 0,C 180,E1 -9603.373,E2 -9603.373} C_VEL
LIN {X 0,Y 432.367,Z 176.127,A -85,B 0,C 180,E1 -9606.024,E2 -9606.024} C_VEL
LIN {X 0,Y 432.346,Z 176.127,A -85,B 0,C 180,E1 -9609.046,E2 -9609.046} C_VEL
LIN {X 0,Y 432.374,Z 176.128,A -85,B 0,C 180,E1 -9612.011,E2 -9612.011} C_VEL
LIN {X 0,Y 432.393,Z 176.126,A -85,B 0,C 180,E1 -9614.927,E2 -9614.927} C_VEL
LIN {X 0,Y 432.455,Z 176.116,A -85,B 0,C 180,E1 -9617.804,E2 -9617.804} C_VEL
LIN {X 0,Y 432.488,Z 176.114,A -85,B 0,C 180,E1 -9621.59,E2 -9621.59} C_VEL
LIN {X 0,Y 432.596,Z 176.099,A -85,B 0,C 180,E1 -9624.406,E2 -9624.406} C_VEL
LIN {X 0,Y 432.603,Z 176.097,A -85,B 0,C 180,E1 -9628.138,E2 -9628.138} C_VEL
LIN {X 0,Y 432.731,Z 176.083,A -85,B 0,C 180,E1 -9630,E2 -9630} C_VEL
LIN {X 0,Y 432.602,Z 176.1,A -85,B 0,C 180,E1 -9632.794,E2 -9632.794} C_VEL
LIN {X 0,Y 432.462,Z 176.115,A -85,B 0,C 180,E1 -9635.026,E2 -9635.026} C_VEL
LIN {X 0,Y 431.902,Z 176.185,A -85,B 0,C 180,E1 -9635.805,E2 -9635.805} C_VEL
LIN {X 0,Y 429.056,Z 176.542,A -85,B 0,C 180,E1 -9637.069,E2 -9637.069} C_VEL
LIN {X 0,Y 426.572,Z 176.85,A -85,B 0,C 180,E1 -9638.09,E2 -9638.09} C_VEL
LIN {X 0,Y 425.491,Z 176.986,A -85,B 0,C 180,E1 -9638.88,E2 -9638.88} C_VEL
LIN {X 0,Y 425.399,Z 176.995,A -85,B 0,C 180,E1 -9639.148,E2 -9639.148} C_VEL
LIN {X 0,Y 425.389,Z 176.999,A -85,B 0,C 180,E1 -9642.904,E2 -9642.904} C_VEL
LIN {X 0,Y 425.357,Z 177.004,A -85,B 0,C 180,E1 -9646.605,E2 -9646.605} C_VEL
LIN {X 0,Y 425.324,Z 177.001,A -85,B 0,C 180,E1 -9649.636,E2 -9649.636} C_VEL
LIN {X 0,Y 425.303,Z 177.003,A -85,B 0,C 180,E1 -9653.365,E2 -9653.365} C_VEL
LIN {X 0,Y 425.343,Z 176.999,A -85,B 0,C 180,E1 -9656.844,E2 -9656.844} C_VEL
LIN {X 0,Y 425.314,Z 177.005,A -85,B 0,C 180,E1 -9659.717,E2 -9659.717} C_VEL
LIN {X 0,Y 425.279,Z 177.006,A -85,B 0,C 180,E1 -9663.048,E2 -9663.048} C_VEL
LIN {X 0,Y 425.28,Z 177.014,A -85,B 0,C 180,E1 -9665.929,E2 -9665.929} C_VEL
LIN {X 0,Y 425.305,Z 177.003,A -85,B 0,C 180,E1 -9669.046,E2 -9669.046} C_VEL
LIN {X 0,Y 425.309,Z 177.007,A -85,B 0,C 180,E1 -9671.962,E2 -9671.962} C_VEL
LIN {X 0,Y 425.278,Z 177.009,A -85,B 0,C 180,E1 -9675.283,E2 -9675.283} C_VEL
LIN {X 0,Y 425.298,Z 177.004,A -85,B 0,C 180,E1 -9678.625,E2 -9678.625} C_VEL
LIN {X 0,Y 425.317,Z 177.005,A -85,B 0,C 180,E1 -9681.104,E2 -9681.104} C_VEL
LIN {X 0,Y 425.294,Z 177.005,A -85,B 0,C 180,E1 -9684.664,E2 -9684.664} C_VEL
LIN {X 0,Y 425.259,Z 177.009,A -85,B 0,C 180,E1 -9688.073,E2 -9688.073} C_VEL
LIN {X 0,Y 425.331,Z 177.005,A -85,B 0,C 180,E1 -9691.369,E2 -9691.369} C_VEL
LIN {X 0,Y 425.289,Z 177.007,A -85,B 0,C 180,E1 -9694.555,E2 -9694.555} C_VEL
LIN {X 0,Y 425.281,Z 177.007,A -85,B 0,C 180,E1 -9697.662,E2 -9697.662} C_VEL
LIN {X 0,Y 425.356,Z 177.002,A -85,B 0,C 180,E1 -9700.704,E2 -9700.704} C_VEL
LIN {X 0,Y 425.382,Z 176.994,A -85,B 0,C 180,E1 -9703.689,E2 -9703.689} C_VEL
LIN {X 0,Y 425.406,Z 176.991,A -85,B 0,C 180,E1 -9707.599,E2 -9707.599} C_VEL
LIN {X 0,Y 425.436,Z 176.987,A -85,B 0,C 180,E1 -9711.45,E2 -9711.45} C_VEL
LIN {X 0,Y 425.547,Z 176.978,A -85,B 0,C 180,E1 -9714.314,E2 -9714.314} C_VEL
LIN {X 0,Y 425.567,Z 176.975,A -85,B 0,C 180,E1 -9718.108,E2 -9718.108} C_VEL
LIN {X 0,Y 425.697,Z 176.958,A -85,B 0,C 180,E1 -9720.001,E2 -9720.001} C_VEL
LIN {X 0,Y 425.539,Z 176.975,A -85,B 0,C 180,E1 -9722.84,E2 -9722.84} C_VEL
LIN {X 0,Y 425.518,Z 176.978,A -85,B 0,C 180,E1 -9726.64,E2 -9726.64} C_VEL
LIN {X 0,Y 425.396,Z 176.994,A -85,B 0,C 180,E1 -9729.51,E2 -9729.51} C_VEL
LIN {X 0,Y 425.389,Z 176.993,A -85,B 0,C 180,E1 -9732.904,E2 -9732.904} C_VEL
LIN {X 0,Y 425.357,Z 176.997,A -85,B 0,C 180,E1 -9736.606,E2 -9736.606} C_VEL
LIN {X 0,Y 425.324,Z 177.007,A -85,B 0,C 180,E1 -9739.636,E2 -9739.636} C_VEL
LIN {X 0,Y 425.303,Z 177.008,A -85,B 0,C 180,E1 -9743.366,E2 -9743.366} C_VEL
LIN {X 0,Y 425.344,Z 176.999,A -85,B 0,C 180,E1 -9746.845,E2 -9746.845} C_VEL
LIN {X 0,Y 425.287,Z 177.009,A -85,B 0,C 180,E1 -9749.72,E2 -9749.72} C_VEL
LIN {X 0,Y 425.28,Z 177.01,A -85,B 0,C 180,E1 -9753.049,E2 -9753.049} C_VEL
LIN {X 0,Y 425.28,Z 177.011,A -85,B 0,C 180,E1 -9755.929,E2 -9755.929} C_VEL
LIN {X 0,Y 425.28,Z 177.013,A -85,B 0,C 180,E1 -9759.042,E2 -9759.042} C_VEL
LIN {X 0,Y 425.325,Z 177.231,A -85,B 0,C 180,E1 -9760.528,E2 -9760.528} C_VEL
LIN {X 0,Y 425.825,Z 180.664,A -85,B 0,C 180,E1 -9763.883,E2 -9763.883} C_VEL
LIN {X 0,Y 426.256,Z 183.567,A -85,B 0,C 180,E1 -9766.508,E2 -9766.508} C_VEL
LIN {X 0,Y 426.381,Z 186.967,A -85,B 0,C 180,E1 -9769.308,E2 -9769.308} C_VEL
LIN {X 0,Y 426.058,Z 191.058,A -85,B 0,C 180,E1 -9772.387,E2 -9772.387} C_VEL
LIN {X 0,Y 425.678,Z 195.945,A -85,B 0,C 180,E1 -9775.852,E2 -9775.852} C_VEL
LIN {X 0,Y 425.296,Z 201.025,A -85,B 0,C 180,E1 -9779.239,E2 -9779.239} C_VEL
LIN {X 0,Y 425.024,Z 206.039,A -85,B 0,C 180,E1 -9782.42,E2 -9782.42} C_VEL
LIN {X 0,Y 424.761,Z 211.212,A -85,B 0,C 180,E1 -9785.566,E2 -9785.566} C_VEL
LIN {X 0,Y 424.579,Z 216.453,A -85,B 0,C 180,E1 -9788.644,E2 -9788.644} C_VEL
LIN {X 0,Y 424.361,Z 221.712,A -85,B 0,C 180,E1 -9791.66,E2 -9791.66} C_VEL
LIN {X 0,Y 424.314,Z 224.163,A -85,B 0,C 180,E1 -9793.019,E2 -9793.019} C_VEL
LIN {X 0,Y 427.085,Z 238.92,A -85,B 0,C 180,E1 -9793.607,E2 -9793.607} C_VEL
LIN {X 0,Y 428.698,Z 249.897,A -85,B 0,C 180,E1 -9794.184,E2 -9794.184} C_VEL
LIN {X 0,Y 428.014,Z 261.45,A -85,B 0,C 180,E1 -9794.891,E2 -9794.891} C_VEL
LIN {X 0,Y 427.471,Z 270.731,A -85,B 0,C 180,E1 -9795.602,E2 -9795.602} C_VEL
LIN {X 0,Y 426.949,Z 279.164,A -85,B 0,C 180,E1 -9796.379,E2 -9796.379} C_VEL
LIN {X 0,Y 426.419,Z 288.218,A -85,B 0,C 180,E1 -9797.386,E2 -9797.386} C_VEL
LIN {X 0,Y 425.876,Z 295.439,A -85,B 0,C 180,E1 -9798.337,E2 -9798.337} C_VEL
LIN {X 0,Y 425.439,Z 301.644,A -85,B 0,C 180,E1 -9799.29,E2 -9799.29} C_VEL
LIN {X 0,Y 425.025,Z 308.185,A -85,B 0,C 180,E1 -9800.482,E2 -9800.482} C_VEL
LIN {X 0,Y 424.737,Z 312.688,A -85,B 0,C 180,E1 -9801.436,E2 -9801.436} C_VEL
LIN {X 0,Y 424.44,Z 318.181,A -85,B 0,C 180,E1 -9802.866,E2 -9802.866} C_VEL
LIN {X 0,Y 424.251,Z 322.506,A -85,B 0,C 180,E1 -9804.296,E2 -9804.296} C_VEL
LIN {X 0,Y 424.221,Z 324.873,A -85,B 0,C 180,E1 -9805.249,E2 -9805.249} C_VEL
LIN {X 0,Y 424.127,Z 328.057,A -85,B 0,C 180,E1 -9807.151,E2 -9807.151} C_VEL
LIN {X 0,Y 424.126,Z 329.115,A -85,B 0,C 180,E1 -9808.101,E2 -9808.101} C_VEL
LIN {X 0,Y 424.069,Z 329.702,A -85,B 0,C 180,E1 -9809.05,E2 -9809.05} C_VEL
LIN {X 0,Y 424.069,Z 329.702,A -85,B 0,C 180,E1 -9810.95,E2 -9810.95} C_VEL
LIN {X 0,Y 424.126,Z 329.115,A -85,B 0,C 180,E1 -9811.899,E2 -9811.899} C_VEL
LIN {X 0,Y 424.11,Z 326.67,A -85,B 0,C 180,E1 -9813.801,E2 -9813.801} C_VEL
LIN {X 0,Y 424.246,Z 323.724,A -85,B 0,C 180,E1 -9815.228,E2 -9815.228} C_VEL
LIN {X 0,Y 424.361,Z 319.735,A -85,B 0,C 180,E1 -9816.657,E2 -9816.657} C_VEL
LIN {X 0,Y 424.59,Z 314.603,A -85,B 0,C 180,E1 -9818.088,E2 -9818.088} C_VEL
LIN {X 0,Y 424.925,Z 309.34,A -85,B 0,C 180,E1 -9819.28,E2 -9819.28} C_VEL
LIN {X 0,Y 425.329,Z 303.02,A -85,B 0,C 180,E1 -9820.472,E2 -9820.472} C_VEL
LIN {X 0,Y 425.723,Z 297.066,A -85,B 0,C 180,E1 -9821.426,E2 -9821.426} C_VEL
LIN {X 0,Y 426.272,Z 290.137,A -85,B 0,C 180,E1 -9822.376,E2 -9822.376} C_VEL
LIN {X 0,Y 426.793,Z 281.953,A -85,B 0,C 180,E1 -9823.329,E2 -9823.329} C_VEL
LIN {X 0,Y 427.221,Z 273.954,A -85,B 0,C 180,E1 -9824.117,E2 -9824.117} C_VEL
LIN {X 0,Y 427.838,Z 264.716,A -85,B 0,C 180,E1 -9824.872,E2 -9824.872} C_VEL
LIN {X 0,Y 428.378,Z 255.963,A -85,B 0,C 180,E1 -9825.462,E2 -9825.462} C_VEL
LIN {X 0,Y 428.571,Z 248.727,A -85,B 0,C 180,E1 -9825.881,E2 -9825.881} C_VEL
LIN {X 0,Y 426.594,Z 236.317,A -85,B 0,C 180,E1 -9826.504,E2 -9826.504} C_VEL
LIN {X 0,Y 424.475,Z 225.445,A -85,B 0,C 180,E1 -9826.922,E2 -9826.922} C_VEL
LIN {X 0,Y 424.314,Z 224.162,A -85,B 0,C 180,E1 -9826.981,E2 -9826.981} C_VEL
LIN {X 0,Y 424.489,Z 218.189,A -85,B 0,C 180,E1 -9830.345,E2 -9830.345} C_VEL
LIN {X 0,Y 424.666,Z 212.939,A -85,B 0,C 180,E1 -9833.402,E2 -9833.402} C_VEL
LIN {X 0,Y 424.969,Z 207.38,A -85,B 0,C 180,E1 -9836.742,E2 -9836.742} C_VEL
LIN {X 0,Y 425.189,Z 202.626,A -85,B 0,C 180,E1 -9839.727,E2 -9839.727} C_VEL
LIN {X 0,Y 425.508,Z 197.588,A -85,B 0,C 180,E1 -9843.028,E2 -9843.028} C_VEL
LIN {X 0,Y 425.852,Z 193.234,A -85,B 0,C 180,E1 -9846.034,E2 -9846.034} C_VEL
LIN {X 0,Y 426.255,Z 188.913,A -85,B 0,C 180,E1 -9849.201,E2 -9849.201} C_VEL
LIN {X 0,Y 426.367,Z 185.195,A -85,B 0,C 180,E1 -9852.118,E2 -9852.118} C_VEL
LIN {X 0,Y 426.057,Z 182.071,A -85,B 0,C 180,E1 -9854.821,E2 -9854.821} C_VEL
LIN {X 0,Y 425.513,Z 178.683,A -85,B 0,C 180,E1 -9858.008,E2 -9858.008} C_VEL
LIN {X 0,Y 425.283,Z 177.013,A -85,B 0,C 180,E1 -9859.872,E2 -9859.872} C_VEL
LIN {X 0,Y 425.275,Z 177.013,A -85,B 0,C 180,E1 -9862.488,E2 -9862.488} C_VEL
LIN {X 0,Y 425.305,Z 177.004,A -85,B 0,C 180,E1 -9865.817,E2 -9865.817} C_VEL
LIN {X 0,Y 425.288,Z 177.006,A -85,B 0,C 180,E1 -9869.238,E2 -9869.238} C_VEL
LIN {X 0,Y 425.345,Z 177.005,A -85,B 0,C 180,E1 -9872.442,E2 -9872.442} C_VEL
LIN {X 0,Y 425.348,Z 176.998,A -85,B 0,C 180,E1 -9875.601,E2 -9875.601} C_VEL
LIN {X 0,Y 425.289,Z 177.008,A -85,B 0,C 180,E1 -9878.681,E2 -9878.681} C_VEL
LIN {X 0,Y 425.328,Z 177.002,A -85,B 0,C 180,E1 -9881.702,E2 -9881.702} C_VEL
LIN {X 0,Y 425.343,Z 177,A -85,B 0,C 180,E1 -9884.67,E2 -9884.67} C_VEL
LIN {X 0,Y 425.407,Z 176.993,A -85,B 0,C 180,E1 -9887.598,E2 -9887.598} C_VEL
LIN {X 0,Y 425.437,Z 176.989,A -85,B 0,C 180,E1 -9891.449,E2 -9891.449} C_VEL
LIN {X 0,Y 425.545,Z 176.975,A -85,B 0,C 180,E1 -9894.313,E2 -9894.313} C_VEL
LIN {X 0,Y 425.566,Z 176.974,A -85,B 0,C 180,E1 -9898.107,E2 -9898.107} C_VEL
LIN {X 0,Y 425.697,Z 176.958,A -85,B 0,C 180,E1 -9899.999,E2 -9899.999} C_VEL
LIN {X 0,Y 425.54,Z 176.974,A -85,B 0,C 180,E1 -9902.839,E2 -9902.839} C_VEL
LIN {X 0,Y 425.523,Z 176.976,A -85,B 0,C 180,E1 -9906.643,E2 -9906.643} C_VEL
LIN {X 0,Y 425.395,Z 176.998,A -85,B 0,C 180,E1 -9909.509,E2 -9909.509} C_VEL
LIN {X 0,Y 425.387,Z 176.996,A -85,B 0,C 180,E1 -9912.903,E2 -9912.903} C_VEL
LIN {X 0,Y 425.355,Z 176.998,A -85,B 0,C 180,E1 -9916.605,E2 -9916.605} C_VEL
LIN {X 0,Y 425.322,Z 177.003,A -85,B 0,C 180,E1 -9919.635,E2 -9919.635} C_VEL
LIN {X 0,Y 425.3,Z 177.007,A -85,B 0,C 180,E1 -9923.365,E2 -9923.365} C_VEL
LIN {X 0,Y 425.342,Z 177.006,A -85,B 0,C 180,E1 -9926.844,E2 -9926.844} C_VEL
LIN {X 0,Y 425.312,Z 177.002,A -85,B 0,C 180,E1 -9929.717,E2 -9929.717} C_VEL
LIN {X 0,Y 425.276,Z 177.01,A -85,B 0,C 180,E1 -9933.048,E2 -9933.048} C_VEL
LIN {X 0,Y 425.278,Z 177.007,A -85,B 0,C 180,E1 -9935.929,E2 -9935.929} C_VEL
LIN {X 0,Y 425.306,Z 177.005,A -85,B 0,C 180,E1 -9939.046,E2 -9939.046} C_VEL
LIN {X 0,Y 425.309,Z 177.005,A -85,B 0,C 180,E1 -9941.962,E2 -9941.962} C_VEL
LIN {X 0,Y 425.279,Z 177.006,A -85,B 0,C 180,E1 -9945.283,E2 -9945.283} C_VEL
LIN {X 0,Y 425.269,Z 177.01,A -85,B 0,C 180,E1 -9948.622,E2 -9948.622} C_VEL
LIN {X 0,Y 425.31,Z 177.003,A -85,B 0,C 180,E1 -9951.103,E2 -9951.103} C_VEL
LIN {X 0,Y 425.295,Z 177.005,A -85,B 0,C 180,E1 -9954.664,E2 -9954.664} C_VEL
LIN {X 0,Y 425.268,Z 177.014,A -85,B 0,C 180,E1 -9958.074,E2 -9958.074} C_VEL
LIN {X 0,Y 425.333,Z 177.002,A -85,B 0,C 180,E1 -9961.369,E2 -9961.369} C_VEL
LIN {X 0,Y 425.291,Z 177.005,A -85,B 0,C 180,E1 -9964.555,E2 -9964.555} C_VEL
LIN {X 0,Y 425.284,Z 177.013,A -85,B 0,C 180,E1 -9967.661,E2 -9967.661} C_VEL
LIN {X 0,Y 425.358,Z 176.997,A -85,B 0,C 180,E1 -9970.704,E2 -9970.704} C_VEL
LIN {X 0,Y 425.385,Z 176.999,A -85,B 0,C 180,E1 -9973.688,E2 -9973.688} C_VEL
LIN {X 0,Y 425.408,Z 176.996,A -85,B 0,C 180,E1 -9977.598,E2 -9977.598} C_VEL
LIN {X 0,Y 425.439,Z 176.992,A -85,B 0,C 180,E1 -9981.45,E2 -9981.45} C_VEL
LIN {X 0,Y 425.552,Z 176.976,A -85,B 0,C 180,E1 -9984.313,E2 -9984.313} C_VEL
LIN {X 0,Y 425.572,Z 176.973,A -85,B 0,C 180,E1 -9988.107,E2 -9988.107} C_VEL
LIN {X 0,Y 425.7,Z 176.959,A -85,B 0,C 180,E1 -9990,E2 -9990} C_VEL
LIN {X 0,Y 425.554,Z 176.978,A -85,B 0,C 180,E1 -9992.84,E2 -9992.84} C_VEL
LIN {X 0,Y 425.528,Z 176.981,A -85,B 0,C 180,E1 -9996.639,E2 -9996.639} C_VEL
LIN {X 0,Y 425.399,Z 176.995,A -85,B 0,C 180,E1 -9999.148,E2 -9999.148} C_VEL
LIN {X 0,Y 424.727,Z 177.081,A -85,B 0,C 180,E1 -9999.938,E2 -9999.938} C_VEL
LIN {X 0,Y 421.879,Z 177.437,A -85,B 0,C 180,E1 -10001.222,E2 -10001.222} C_VEL
LIN {X 0,Y 419.463,Z 177.738,A -85,B 0,C 180,E1 -10002.258,E2 -10002.258} C_VEL
LIN {X 0,Y 418.412,Z 177.868,A -85,B 0,C 180,E1 -10003.058,E2 -10003.058} C_VEL
LIN {X 0,Y 418.319,Z 177.878,A -85,B 0,C 180,E1 -10003.33,E2 -10003.33} C_VEL
LIN {X 0,Y 418.309,Z 177.881,A -85,B 0,C 180,E1 -10006.736,E2 -10006.736} C_VEL
LIN {X 0,Y 418.267,Z 177.881,A -85,B 0,C 180,E1 -10009.79,E2 -10009.79} C_VEL
LIN {X 0,Y 418.234,Z 177.887,A -85,B 0,C 180,E1 -10012.736,E2 -10012.736} C_VEL
LIN {X 0,Y 418.266,Z 177.883,A -85,B 0,C 180,E1 -10015.904,E2 -10015.904} C_VEL
LIN {X 0,Y 418.27,Z 177.88,A -85,B 0,C 180,E1 -10019.161,E2 -10019.161} C_VEL
LIN {X 0,Y 418.255,Z 177.882,A -85,B 0,C 180,E1 -10022.845,E2 -10022.845} C_VEL
LIN {X 0,Y 418.243,Z 177.886,A -85,B 0,C 180,E1 -10026.239,E2 -10026.239} C_VEL
LIN {X 0,Y 418.258,Z 177.887,A -85,B 0,C 180,E1 -10029.68,E2 -10029.68} C_VEL
LIN {X 0,Y 418.24,Z 177.884,A -85,B 0,C 180,E1 -10032.324,E2 -10032.324} C_VEL
LIN {X 0,Y 418.229,Z 177.886,A -85,B 0,C 180,E1 -10035.109,E2 -10035.109} C_VEL
LIN {X 0,Y 418.25,Z 177.887,A -85,B 0,C 180,E1 -10037.769,E2 -10037.769} C_VEL
LIN {X 0,Y 418.262,Z 177.881,A -85,B 0,C 180,E1 -10040.617,E2 -10040.617} C_VEL
LIN {X 0,Y 418.24,Z 177.885,A -85,B 0,C 180,E1 -10043.976,E2 -10043.976} C_VEL
LIN {X 0,Y 418.251,Z 177.887,A -85,B 0,C 180,E1 -10047.156,E2 -10047.156} C_VEL
LIN {X 0,Y 418.268,Z 177.883,A -85,B 0,C 180,E1 -10050.839,E2 -10050.839} C_VEL
LIN {X 0,Y 418.264,Z 177.88,A -85,B 0,C 180,E1 -10054.096,E2 -10054.096} C_VEL
LIN {X 0,Y 418.232,Z 177.888,A -85,B 0,C 180,E1 -10057.264,E2 -10057.264} C_VEL
LIN {X 0,Y 418.277,Z 177.88,A -85,B 0,C 180,E1 -10060.364,E2 -10060.364} C_VEL
LIN {X 0,Y 418.311,Z 177.876,A -85,B 0,C 180,E1 -10063.405,E2 -10063.405} C_VEL
LIN {X 0,Y 418.34,Z 177.874,A -85,B 0,C 180,E1 -10067,E2 -10067} C_VEL
LIN {X 0,Y 418.335,Z 177.875,A -85,B 0,C 180,E1 -10070.329,E2 -10070.329} C_VEL
LIN {X 0,Y 418.486,Z 177.853,A -85,B 0,C 180,E1 -10073.249,E2 -10073.249} C_VEL
LIN {X 0,Y 418.333,Z 177.872,A -85,B 0,C 180,E1 -10075.182,E2 -10075.182} C_VEL
LIN {X 0,Y 418.537,Z 177.85,A -85,B 0,C 180,E1 -10078.076,E2 -10078.076} C_VEL
LIN {X 0,Y 418.666,Z 177.834,A -85,B 0,C 180,E1 -10080.001,E2 -10080.001} C_VEL
LIN {X 0,Y 418.495,Z 177.852,A -85,B 0,C 180,E1 -10082.888,E2 -10082.888} C_VEL
LIN {X 0,Y 418.482,Z 177.854,A -85,B 0,C 180,E1 -10086.752,E2 -10086.752} C_VEL
LIN {X 0,Y 418.336,Z 177.874,A -85,B 0,C 180,E1 -10089.672,E2 -10089.672} C_VEL
LIN {X 0,Y 418.342,Z 177.871,A -85,B 0,C 180,E1 -10093.001,E2 -10093.001} C_VEL
LIN {X 0,Y 418.309,Z 177.875,A -85,B 0,C 180,E1 -10096.736,E2 -10096.736} C_VEL
LIN {X 0,Y 418.267,Z 177.886,A -85,B 0,C 180,E1 -10099.791,E2 -10099.791} C_VEL
LIN {X 0,Y 418.235,Z 177.884,A -85,B 0,C 180,E1 -10102.737,E2 -10102.737} C_VEL
LIN {X 0,Y 418.268,Z 177.883,A -85,B 0,C 180,E1 -10105.905,E2 -10105.905} C_VEL
LIN {X 0,Y 418.262,Z 177.884,A -85,B 0,C 180,E1 -10109.163,E2 -10109.163} C_VEL
LIN {X 0,Y 418.255,Z 177.883,A -85,B 0,C 180,E1 -10112.845,E2 -10112.845} C_VEL
LIN {X 0,Y 418.242,Z 177.887,A -85,B 0,C 180,E1 -10116.239,E2 -10116.239} C_VEL
LIN {X 0,Y 418.243,Z 177.889,A -85,B 0,C 180,E1 -10119.683,E2 -10119.683} C_VEL
LIN {X 0,Y 418.597,Z 180.263,A -85,B 0,C 180,E1 -10122.377,E2 -10122.377} C_VEL
LIN {X 0,Y 419.062,Z 183.243,A -85,B 0,C 180,E1 -10125.222,E2 -10125.222} C_VEL
LIN {X 0,Y 419.379,Z 186.322,A -85,B 0,C 180,E1 -10127.909,E2 -10127.909} C_VEL
LIN {X 0,Y 419.278,Z 189.486,A -85,B 0,C 180,E1 -10130.45,E2 -10130.45} C_VEL
LIN {X 0,Y 418.868,Z 193.746,A -85,B 0,C 180,E1 -10133.647,E2 -10133.647} C_VEL
LIN {X 0,Y 418.447,Z 198.678,A -85,B 0,C 180,E1 -10137.117,E2 -10137.117} C_VEL
LIN {X 0,Y 418.177,Z 202.563,A -85,B 0,C 180,E1 -10139.723,E2 -10139.723} C_VEL
LIN {X 0,Y 417.929,Z 207.711,A -85,B 0,C 180,E1 -10143.033,E2 -10143.033} C_VEL
LIN {X 0,Y 417.609,Z 212.814,A -85,B 0,C 180,E1 -10146.178,E2 -10146.178} C_VEL
LIN {X 0,Y 417.515,Z 216.309,A -85,B 0,C 180,E1 -10148.265,E2 -10148.265} C_VEL
LIN {X 0,Y 417.312,Z 221.553,A -85,B 0,C 180,E1 -10151.339,E2 -10151.339} C_VEL
LIN {X 0,Y 417.25,Z 223.992,A -85,B 0,C 180,E1 -10152.73,E2 -10152.73} C_VEL
LIN {X 0,Y 419.797,Z 237.424,A -85,B 0,C 180,E1 -10153.268,E2 -10153.268} C_VEL
LIN {X 0,Y 421.758,Z 250.254,A -85,B 0,C 180,E1 -10153.951,E2 -10153.951} C_VEL
LIN {X 0,Y 421.157,Z 261.239,A -85,B 0,C 180,E1 -10154.639,E2 -10154.639} C_VEL
LIN {X 0,Y 420.569,Z 270.519,A -85,B 0,C 180,E1 -10155.36,E2 -10155.36} C_VEL
LIN {X 0,Y 419.957,Z 279.841,A -85,B 0,C 180,E1 -10156.244,E2 -10156.244} C_VEL
LIN {X 0,Y 419.455,Z 288.005,A -85,B 0,C 180,E1 -10157.173,E2 -10157.173} C_VEL
LIN {X 0,Y 418.912,Z 295.228,A -85,B 0,C 180,E1 -10158.141,E2 -10158.141} C_VEL
LIN {X 0,Y 418.41,Z 301.431,A -85,B 0,C 180,E1 -10159.108,E2 -10159.108} C_VEL
LIN {X 0,Y 417.975,Z 307.972,A -85,B 0,C 180,E1 -10160.32,E2 -10160.32} C_VEL
LIN {X 0,Y 417.695,Z 312.476,A -85,B 0,C 180,E1 -10161.29,E2 -10161.29} C_VEL
LIN {X 0,Y 417.366,Z 317.969,A -85,B 0,C 180,E1 -10162.745,E2 -10162.745} C_VEL
LIN {X 0,Y 417.163,Z 322.294,A -85,B 0,C 180,E1 -10164.199,E2 -10164.199} C_VEL
LIN {X 0,Y 417.152,Z 324.662,A -85,B 0,C 180,E1 -10165.168,E2 -10165.168} C_VEL
LIN {X 0,Y 417.025,Z 327.846,A -85,B 0,C 180,E1 -10167.102,E2 -10167.102} C_VEL
LIN {X 0,Y 417.053,Z 328.904,A -85,B 0,C 180,E1 -10168.069,E2 -10168.069} C_VEL
LIN {X 0,Y 416.993,Z 329.491,A -85,B 0,C 180,E1 -10169.034,E2 -10169.034} C_VEL
LIN {X 0,Y 416.993,Z 329.491,A -85,B 0,C 180,E1 -10170.966,E2 -10170.966} C_VEL
LIN {X 0,Y 417.053,Z 328.904,A -85,B 0,C 180,E1 -10171.931,E2 -10171.931} C_VEL
LIN {X 0,Y 417.026,Z 326.458,A -85,B 0,C 180,E1 -10173.865,E2 -10173.865} C_VEL
LIN {X 0,Y 417.164,Z 323.512,A -85,B 0,C 180,E1 -10175.317,E2 -10175.317} C_VEL
LIN {X 0,Y 417.277,Z 319.522,A -85,B 0,C 180,E1 -10176.771,E2 -10176.771} C_VEL
LIN {X 0,Y 417.55,Z 314.392,A -85,B 0,C 180,E1 -10178.225,E2 -10178.225} C_VEL
LIN {X 0,Y 417.893,Z 309.128,A -85,B 0,C 180,E1 -10179.437,E2 -10179.437} C_VEL
LIN {X 0,Y 418.307,Z 302.808,A -85,B 0,C 180,E1 -10180.65,E2 -10180.65} C_VEL
LIN {X 0,Y 418.754,Z 296.854,A -85,B 0,C 180,E1 -10181.618,E2 -10181.618} C_VEL
LIN {X 0,Y 419.303,Z 289.925,A -85,B 0,C 180,E1 -10182.585,E2 -10182.585} C_VEL
LIN {X 0,Y 419.867,Z 281.741,A -85,B 0,C 180,E1 -10183.553,E2 -10183.553} C_VEL
LIN {X 0,Y 420.37,Z 272.924,A -85,B 0,C 180,E1 -10184.427,E2 -10184.427} C_VEL
LIN {X 0,Y 420.951,Z 264.504,A -85,B 0,C 180,E1 -10185.121,E2 -10185.121} C_VEL
LIN {X 0,Y 421.533,Z 255.974,A -85,B 0,C 180,E1 -10185.706,E2 -10185.706} C_VEL
LIN {X 0,Y 421.643,Z 249.241,A -85,B 0,C 180,E1 -10186.112,E2 -10186.112} C_VEL
LIN {X 0,Y 419.561,Z 236.339,A -85,B 0,C 180,E1 -10186.78,E2 -10186.78} C_VEL
LIN {X 0,Y 417.461,Z 225.572,A -85,B 0,C 180,E1 -10187.207,E2 -10187.207} C_VEL
LIN {X 0,Y 417.249,Z 223.992,A -85,B 0,C 180,E1 -10187.27,E2 -10187.27} C_VEL
LIN {X 0,Y 417.436,Z 218.031,A -85,B 0,C 180,E1 -10190.705,E2 -10190.705} C_VEL
LIN {X 0,Y 417.56,Z 214.532,A -85,B 0,C 180,E1 -10192.775,E2 -10192.775} C_VEL
LIN {X 0,Y 417.782,Z 209.362,A -85,B 0,C 180,E1 -10195.936,E2 -10195.936} C_VEL
LIN {X 0,Y 418.091,Z 204.242,A -85,B 0,C 180,E1 -10199.175,E2 -10199.175} C_VEL
LIN {X 0,Y 418.414,Z 199.203,A -85,B 0,C 180,E1 -10202.513,E2 -10202.513} C_VEL
LIN {X 0,Y 418.798,Z 194.282,A -85,B 0,C 180,E1 -10205.968,E2 -10205.968} C_VEL
LIN {X 0,Y 419.107,Z 191.059,A -85,B 0,C 180,E1 -10208.348,E2 -10208.348} C_VEL
LIN {X 0,Y 419.371,Z 187.576,A -85,B 0,C 180,E1 -10211.05,E2 -10211.05} C_VEL
LIN {X 0,Y 419.204,Z 184.26,A -85,B 0,C 180,E1 -10213.871,E2 -10213.871} C_VEL
LIN {X 0,Y 418.745,Z 181.389,A -85,B 0,C 180,E1 -10216.518,E2 -10216.518} C_VEL
LIN {X 0,Y 418.383,Z 178.784,A -85,B 0,C 180,E1 -10219.104,E2 -10219.104} C_VEL
LIN {X 0,Y 418.244,Z 177.889,A -85,B 0,C 180,E1 -10220.62,E2 -10220.62} C_VEL
LIN {X 0,Y 418.24,Z 177.884,A -85,B 0,C 180,E1 -10223.975,E2 -10223.975} C_VEL
LIN {X 0,Y 418.255,Z 177.883,A -85,B 0,C 180,E1 -10227.155,E2 -10227.155} C_VEL
LIN {X 0,Y 418.265,Z 177.883,A -85,B 0,C 180,E1 -10230.895,E2 -10230.895} C_VEL
LIN {X 0,Y 418.268,Z 177.883,A -85,B 0,C 180,E1 -10234.095,E2 -10234.095} C_VEL
LIN {X 0,Y 418.235,Z 177.884,A -85,B 0,C 180,E1 -10237.263,E2 -10237.263} C_VEL
LIN {X 0,Y 418.279,Z 177.885,A -85,B 0,C 180,E1 -10240.363,E2 -10240.363} C_VEL
LIN {X 0,Y 418.313,Z 177.875,A -85,B 0,C 180,E1 -10243.404,E2 -10243.404} C_VEL
LIN {X 0,Y 418.342,Z 177.871,A -85,B 0,C 180,E1 -10246.999,E2 -10246.999} C_VEL
LIN {X 0,Y 418.336,Z 177.874,A -85,B 0,C 180,E1 -10250.328,E2 -10250.328} C_VEL
LIN {X 0,Y 418.482,Z 177.854,A -85,B 0,C 180,E1 -10253.248,E2 -10253.248} C_VEL
LIN {X 0,Y 418.332,Z 177.873,A -85,B 0,C 180,E1 -10255.181,E2 -10255.181} C_VEL
LIN {X 0,Y 418.536,Z 177.85,A -85,B 0,C 180,E1 -10258.075,E2 -10258.075} C_VEL
LIN {X 0,Y 418.666,Z 177.834,A -85,B 0,C 180,E1 -10259.999,E2 -10259.999} C_VEL
LIN {X 0,Y 418.495,Z 177.852,A -85,B 0,C 180,E1 -10262.887,E2 -10262.887} C_VEL
LIN {X 0,Y 418.486,Z 177.853,A -85,B 0,C 180,E1 -10266.751,E2 -10266.751} C_VEL
LIN {X 0,Y 418.335,Z 177.875,A -85,B 0,C 180,E1 -10269.671,E2 -10269.671} C_VEL
LIN {X 0,Y 418.34,Z 177.874,A -85,B 0,C 180,E1 -10273,E2 -10273} C_VEL
LIN {X 0,Y 418.307,Z 177.877,A -85,B 0,C 180,E1 -10276.735,E2 -10276.735} C_VEL
LIN {X 0,Y 418.264,Z 177.881,A -85,B 0,C 180,E1 -10279.79,E2 -10279.79} C_VEL
LIN {X 0,Y 418.232,Z 177.888,A -85,B 0,C 180,E1 -10282.736,E2 -10282.736} C_VEL
LIN {X 0,Y 418.264,Z 177.88,A -85,B 0,C 180,E1 -10285.904,E2 -10285.904} C_VEL
LIN {X 0,Y 418.268,Z 177.883,A -85,B 0,C 180,E1 -10289.161,E2 -10289.161} C_VEL
LIN {X 0,Y 418.251,Z 177.887,A -85,B 0,C 180,E1 -10292.844,E2 -10292.844} C_VEL
LIN {X 0,Y 418.242,Z 177.886,A -85,B 0,C 180,E1 -10296.239,E2 -10296.239} C_VEL
LIN {X 0,Y 418.259,Z 177.881,A -85,B 0,C 180,E1 -10299.68,E2 -10299.68} C_VEL
LIN {X 0,Y 418.239,Z 177.889,A -85,B 0,C 180,E1 -10302.324,E2 -10302.324} C_VEL
LIN {X 0,Y 418.229,Z 177.885,A -85,B 0,C 180,E1 -10305.109,E2 -10305.109} C_VEL
LIN {X 0,Y 418.235,Z 177.886,A -85,B 0,C 180,E1 -10307.767,E2 -10307.767} C_VEL
LIN {X 0,Y 418.254,Z 177.884,A -85,B 0,C 180,E1 -10310.618,E2 -10310.618} C_VEL
LIN {X 0,Y 418.241,Z 177.889,A -85,B 0,C 180,E1 -10313.976,E2 -10313.976} C_VEL
LIN {X 0,Y 418.255,Z 177.882,A -85,B 0,C 180,E1 -10317.155,E2 -10317.155} C_VEL
LIN {X 0,Y 418.27,Z 177.88,A -85,B 0,C 180,E1 -10320.839,E2 -10320.839} C_VEL
LIN {X 0,Y 418.266,Z 177.883,A -85,B 0,C 180,E1 -10324.096,E2 -10324.096} C_VEL
LIN {X 0,Y 418.234,Z 177.887,A -85,B 0,C 180,E1 -10327.264,E2 -10327.264} C_VEL
LIN {X 0,Y 418.279,Z 177.881,A -85,B 0,C 180,E1 -10330.364,E2 -10330.364} C_VEL
LIN {X 0,Y 418.313,Z 177.881,A -85,B 0,C 180,E1 -10333.405,E2 -10333.405} C_VEL
LIN {X 0,Y 418.342,Z 177.877,A -85,B 0,C 180,E1 -10336.999,E2 -10336.999} C_VEL
LIN {X 0,Y 418.338,Z 177.876,A -85,B 0,C 180,E1 -10340.329,E2 -10340.329} C_VEL
LIN {X 0,Y 418.491,Z 177.857,A -85,B 0,C 180,E1 -10343.249,E2 -10343.249} C_VEL
LIN {X 0,Y 418.338,Z 177.877,A -85,B 0,C 180,E1 -10345.182,E2 -10345.182} C_VEL
LIN {X 0,Y 418.541,Z 177.849,A -85,B 0,C 180,E1 -10348.075,E2 -10348.075} C_VEL
LIN {X 0,Y 418.67,Z 177.835,A -85,B 0,C 180,E1 -10350,E2 -10350} C_VEL
LIN {X 0,Y 418.507,Z 177.855,A -85,B 0,C 180,E1 -10352.888,E2 -10352.888} C_VEL
LIN {X 0,Y 418.491,Z 177.857,A -85,B 0,C 180,E1 -10356.751,E2 -10356.751} C_VEL
LIN {X 0,Y 418.338,Z 177.876,A -85,B 0,C 180,E1 -10359.671,E2 -10359.671} C_VEL
LIN {X 0,Y 418.319,Z 177.878,A -85,B 0,C 180,E1 -10363.33,E2 -10363.33} C_VEL
LIN {X 0,Y 417.626,Z 177.965,A -85,B 0,C 180,E1 -10364.133,E2 -10364.133} C_VEL
LIN {X 0,Y 414.748,Z 178.323,A -85,B 0,C 180,E1 -10365.439,E2 -10365.439} C_VEL
LIN {X 0,Y 412.334,Z 178.626,A -85,B 0,C 180,E1 -10366.493,E2 -10366.493} C_VEL
LIN {X 0,Y 411.312,Z 178.751,A -85,B 0,C 180,E1 -10367.308,E2 -10367.308} C_VEL
LIN {X 0,Y 411.236,Z 178.759,A -85,B 0,C 180,E1 -10367.584,E2 -10367.584} C_VEL
LIN {X 0,Y 411.192,Z 178.762,A -85,B 0,C 180,E1 -10371.034,E2 -10371.034} C_VEL
LIN {X 0,Y 411.223,Z 178.764,A -85,B 0,C 180,E1 -10374.215,E2 -10374.215} C_VEL
LIN {X 0,Y 411.255,Z 178.754,A -85,B 0,C 180,E1 -10377.477,E2 -10377.477} C_VEL
LIN {X 0,Y 411.195,Z 178.761,A -85,B 0,C 180,E1 -10380.847,E2 -10380.847} C_VEL
LIN {X 0,Y 411.201,Z 178.763,A -85,B 0,C 180,E1 -10384.333,E2 -10384.333} C_VEL
LIN {X 0,Y 411.198,Z 178.766,A -85,B 0,C 180,E1 -10387.973,E2 -10387.973} C_VEL
LIN {X 0,Y 411.195,Z 178.762,A -85,B 0,C 180,E1 -10391.234,E2 -10391.234} C_VEL
LIN {X 0,Y 411.17,Z 178.764,A -85,B 0,C 180,E1 -10394.49,E2 -10394.49} C_VEL
LIN {X 0,Y 411.192,Z 178.762,A -85,B 0,C 180,E1 -10398.197,E2 -10398.197} C_VEL
LIN {X 0,Y 411.225,Z 178.758,A -85,B 0,C 180,E1 -10400.777,E2 -10400.777} C_VEL
LIN {X 0,Y 411.193,Z 178.761,A -85,B 0,C 180,E1 -10404.472,E2 -10404.472} C_VEL
LIN {X 0,Y 411.201,Z 178.763,A -85,B 0,C 180,E1 -10406.873,E2 -10406.873} C_VEL
LIN {X 0,Y 411.234,Z 178.757,A -85,B 0,C 180,E1 -10410.642,E2 -10410.642} C_VEL
LIN {X 0,Y 411.232,Z 178.758,A -85,B 0,C 180,E1 -10413.619,E2 -10413.619} C_VEL
LIN {X 0,Y 411.197,Z 178.766,A -85,B 0,C 180,E1 -10416.853,E2 -10416.853} C_VEL
LIN {X 0,Y 411.208,Z 178.759,A -85,B 0,C 180,E1 -10420.051,E2 -10420.051} C_VEL
LIN {X 0,Y 411.257,Z 178.757,A -85,B 0,C 180,E1 -10423.131,E2 -10423.131} C_VEL
LIN {X 0,Y 411.299,Z 178.753,A -85,B 0,C 180,E1 -10426.896,E2 -10426.896} C_VEL
LIN {X 0,Y 411.287,Z 178.752,A -85,B 0,C 180,E1 -10430.162,E2 -10430.162} C_VEL
LIN {X 0,Y 411.45,Z 178.73,A -85,B 0,C 180,E1 -10433.133,E2 -10433.133} C_VEL
LIN {X 0,Y 411.304,Z 178.748,A -85,B 0,C 180,E1 -10435.099,E2 -10435.099} C_VEL
LIN {X 0,Y 411.506,Z 178.725,A -85,B 0,C 180,E1 -10438.043,E2 -10438.043} C_VEL
LIN {X 0,Y 411.636,Z 178.709,A -85,B 0,C 180,E1 -10440.001,E2 -10440.001} C_VEL
LIN {X 0,Y 411.452,Z 178.73,A -85,B 0,C 180,E1 -10442.938,E2 -10442.938} C_VEL
LIN {X 0,Y 411.447,Z 178.73,A -85,B 0,C 180,E1 -10446.868,E2 -10446.868} C_VEL
LIN {X 0,Y 411.288,Z 178.754,A -85,B 0,C 180,E1 -10449.839,E2 -10449.839} C_VEL
LIN {X 0,Y 411.301,Z 178.748,A -85,B 0,C 180,E1 -10453.105,E2 -10453.105} C_VEL
LIN {X 0,Y 411.253,Z 178.754,A -85,B 0,C 180,E1 -10456.889,E2 -10456.889} C_VEL
LIN {X 0,Y 411.227,Z 178.761,A -85,B 0,C 180,E1 -10459.987,E2 -10459.987} C_VEL
LIN {X 0,Y 411.2,Z 178.762,A -85,B 0,C 180,E1 -10463.148,E2 -10463.148} C_VEL
LIN {X 0,Y 411.235,Z 178.756,A -85,B 0,C 180,E1 -10466.382,E2 -10466.382} C_VEL
LIN {X 0,Y 411.197,Z 178.764,A -85,B 0,C 180,E1 -10469.713,E2 -10469.713} C_VEL
LIN {X 0,Y 411.204,Z 178.765,A -85,B 0,C 180,E1 -10473.157,E2 -10473.157} C_VEL
LIN {X 0,Y 411.19,Z 178.767,A -85,B 0,C 180,E1 -10476.553,E2 -10476.553} C_VEL
LIN {X 0,Y 411.226,Z 178.89,A -85,B 0,C 180,E1 -10479.731,E2 -10479.731} C_VEL
LIN {X 0,Y 411.719,Z 182.117,A -85,B 0,C 180,E1 -10483.063,E2 -10483.063} C_VEL
LIN {X 0,Y 412.134,Z 184.945,A -85,B 0,C 180,E1 -10485.743,E2 -10485.743} C_VEL
LIN {X 0,Y 412.369,Z 188.188,A -85,B 0,C 180,E1 -10488.582,E2 -10488.582} C_VEL
LIN {X 0,Y 412.164,Z 191.053,A -85,B 0,C 180,E1 -10490.884,E2 -10490.884} C_VEL
LIN {X 0,Y 411.875,Z 194.279,A -85,B 0,C 180,E1 -10493.33,E2 -10493.33} C_VEL
LIN {X 0,Y 411.419,Z 199.165,A -85,B 0,C 180,E1 -10496.864,E2 -10496.864} C_VEL
LIN {X 0,Y 411.07,Z 204.179,A -85,B 0,C 180,E1 -10500.277,E2 -10500.277} C_VEL
LIN {X 0,Y 410.761,Z 209.264,A -85,B 0,C 180,E1 -10503.587,E2 -10503.587} C_VEL
LIN {X 0,Y 410.49,Z 214.42,A -85,B 0,C 180,E1 -10506.81,E2 -10506.81} C_VEL
LIN {X 0,Y 410.365,Z 217.874,A -85,B 0,C 180,E1 -10508.922,E2 -10508.922} C_VEL
LIN {X 0,Y 410.16,Z 223.112,A -85,B 0,C 180,E1 -10512.036,E2 -10512.036} C_VEL
LIN {X 0,Y 410.171,Z 224.001,A -85,B 0,C 180,E1 -10512.445,E2 -10512.445} C_VEL
LIN {X 0,Y 412.189,Z 234.454,A -85,B 0,C 180,E1 -10512.85,E2 -10512.85} C_VEL
LIN {X 0,Y 413.66,Z 242.979,A -85,B 0,C 180,E1 -10513.27,E2 -10513.27} C_VEL
LIN {X 0,Y 414.788,Z 250.623,A -85,B 0,C 180,E1 -10513.71,E2 -10513.71} C_VEL
LIN {X 0,Y 414.301,Z 261.027,A -85,B 0,C 180,E1 -10514.378,E2 -10514.378} C_VEL
LIN {X 0,Y 413.673,Z 270.307,A -85,B 0,C 180,E1 -10515.11,E2 -10515.11} C_VEL
LIN {X 0,Y 413.027,Z 279.629,A -85,B 0,C 180,E1 -10516.009,E2 -10516.009} C_VEL
LIN {X 0,Y 412.497,Z 287.793,A -85,B 0,C 180,E1 -10516.953,E2 -10516.953} C_VEL
LIN {X 0,Y 411.935,Z 295.015,A -85,B 0,C 180,E1 -10517.937,E2 -10517.937} C_VEL
LIN {X 0,Y 411.411,Z 301.219,A -85,B 0,C 180,E1 -10518.92,E2 -10518.92} C_VEL
LIN {X 0,Y 410.944,Z 307.76,A -85,B 0,C 180,E1 -10520.153,E2 -10520.153} C_VEL
LIN {X 0,Y 410.635,Z 312.263,A -85,B 0,C 180,E1 -10521.139,E2 -10521.139} C_VEL
LIN {X 0,Y 410.293,Z 317.756,A -85,B 0,C 180,E1 -10522.619,E2 -10522.619} C_VEL
LIN {X 0,Y 410.086,Z 322.082,A -85,B 0,C 180,E1 -10524.098,E2 -10524.098} C_VEL
LIN {X 0,Y 410.061,Z 324.451,A -85,B 0,C 180,E1 -10525.084,E2 -10525.084} C_VEL
LIN {X 0,Y 409.924,Z 327.634,A -85,B 0,C 180,E1 -10527.052,E2 -10527.052} C_VEL
LIN {X 0,Y 409.964,Z 328.693,A -85,B 0,C 180,E1 -10528.035,E2 -10528.035} C_VEL
LIN {X 0,Y 409.919,Z 329.28,A -85,B 0,C 180,E1 -10529.018,E2 -10529.018} C_VEL
LIN {X 0,Y 409.919,Z 329.28,A -85,B 0,C 180,E1 -10530.982,E2 -10530.982} C_VEL
LIN {X 0,Y 409.964,Z 328.693,A -85,B 0,C 180,E1 -10531.965,E2 -10531.965} C_VEL
LIN {X 0,Y 409.946,Z 326.247,A -85,B 0,C 180,E1 -10533.932,E2 -10533.932} C_VEL
LIN {X 0,Y 410.063,Z 323.3,A -85,B 0,C 180,E1 -10535.409,E2 -10535.409} C_VEL
LIN {X 0,Y 410.2,Z 319.31,A -85,B 0,C 180,E1 -10536.888,E2 -10536.888} C_VEL
LIN {X 0,Y 410.499,Z 314.179,A -85,B 0,C 180,E1 -10538.368,E2 -10538.368} C_VEL
LIN {X 0,Y 410.863,Z 308.916,A -85,B 0,C 180,E1 -10539.6,E2 -10539.6} C_VEL
LIN {X 0,Y 411.284,Z 302.595,A -85,B 0,C 180,E1 -10540.834,E2 -10540.834} C_VEL
LIN {X 0,Y 411.763,Z 296.642,A -85,B 0,C 180,E1 -10541.819,E2 -10541.819} C_VEL
LIN {X 0,Y 412.332,Z 289.712,A -85,B 0,C 180,E1 -10542.802,E2 -10542.802} C_VEL
LIN {X 0,Y 412.955,Z 281.529,A -85,B 0,C 180,E1 -10543.784,E2 -10543.784} C_VEL
LIN {X 0,Y 413.467,Z 272.846,A -85,B 0,C 180,E1 -10544.661,E2 -10544.661} C_VEL
LIN {X 0,Y 414.091,Z 264.292,A -85,B 0,C 180,E1 -10545.378,E2 -10545.378} C_VEL
LIN {X 0,Y 414.772,Z 254.231,A -85,B 0,C 180,E1 -10546.064,E2 -10546.064} C_VEL
LIN {X 0,Y 414.559,Z 248.784,A -85,B 0,C 180,E1 -10546.408,E2 -10546.408} C_VEL
LIN {X 0,Y 412.489,Z 236.009,A -85,B 0,C 180,E1 -10547.081,E2 -10547.081} C_VEL
LIN {X 0,Y 410.363,Z 225.411,A -85,B 0,C 180,E1 -10547.513,E2 -10547.513} C_VEL
LIN {X 0,Y 410.156,Z 223.808,A -85,B 0,C 180,E1 -10547.577,E2 -10547.577} C_VEL
LIN {X 0,Y 410.29,Z 219.595,A -85,B 0,C 180,E1 -10550.034,E2 -10550.034} C_VEL
LIN {X 0,Y 410.493,Z 215.675,A -85,B 0,C 180,E1 -10552.402,E2 -10552.402} C_VEL
LIN {X 0,Y 410.653,Z 210.964,A -85,B 0,C 180,E1 -10555.331,E2 -10555.331} C_VEL
LIN {X 0,Y 410.957,Z 205.848,A -85,B 0,C 180,E1 -10558.609,E2 -10558.609} C_VEL
LIN {X 0,Y 411.272,Z 200.82,A -85,B 0,C 180,E1 -10561.987,E2 -10561.987} C_VEL
LIN {X 0,Y 411.701,Z 195.906,A -85,B 0,C 180,E1 -10565.478,E2 -10565.478} C_VEL
LIN {X 0,Y 412.07,Z 192.077,A -85,B 0,C 180,E1 -10568.321,E2 -10568.321} C_VEL
LIN {X 0,Y 412.358,Z 188.192,A -85,B 0,C 180,E1 -10571.417,E2 -10571.417} C_VEL
LIN {X 0,Y 412.118,Z 184.831,A -85,B 0,C 180,E1 -10574.361,E2 -10574.361} C_VEL
LIN {X 0,Y 411.64,Z 181.823,A -85,B 0,C 180,E1 -10577.234,E2 -10577.234} C_VEL
LIN {X 0,Y 411.227,Z 178.887,A -85,B 0,C 180,E1 -10580.269,E2 -10580.269} C_VEL
LIN {X 0,Y 411.19,Z 178.763,A -85,B 0,C 180,E1 -10583.447,E2 -10583.447} C_VEL
LIN {X 0,Y 411.205,Z 178.764,A -85,B 0,C 180,E1 -10586.873,E2 -10586.873} C_VEL
LIN {X 0,Y 411.23,Z 178.763,A -85,B 0,C 180,E1 -10590.643,E2 -10590.643} C_VEL
LIN {X 0,Y 411.235,Z 178.756,A -85,B 0,C 180,E1 -10593.618,E2 -10593.618} C_VEL
LIN {X 0,Y 411.2,Z 178.762,A -85,B 0,C 180,E1 -10596.852,E2 -10596.852} C_VEL
LIN {X 0,Y 411.211,Z 178.763,A -85,B 0,C 180,E1 -10600.05,E2 -10600.05} C_VEL
LIN {X 0,Y 411.259,Z 178.753,A -85,B 0,C 180,E1 -10603.13,E2 -10603.13} C_VEL
LIN {X 0,Y 411.301,Z 178.748,A -85,B 0,C 180,E1 -10606.895,E2 -10606.895} C_VEL
LIN {X 0,Y 411.288,Z 178.754,A -85,B 0,C 180,E1 -10610.161,E2 -10610.161} C_VEL
LIN {X 0,Y 411.447,Z 178.73,A -85,B 0,C 180,E1 -10613.132,E2 -10613.132} C_VEL
LIN {X 0,Y 411.303,Z 178.748,A -85,B 0,C 180,E1 -10615.098,E2 -10615.098} C_VEL
LIN {X 0,Y 411.505,Z 178.726,A -85,B 0,C 180,E1 -10618.042,E2 -10618.042} C_VEL
LIN {X 0,Y 411.636,Z 178.709,A -85,B 0,C 180,E1 -10619.999,E2 -10619.999} C_VEL
LIN {X 0,Y 411.452,Z 178.73,A -85,B 0,C 180,E1 -10622.937,E2 -10622.937} C_VEL
LIN {X 0,Y 411.45,Z 178.73,A -85,B 0,C 180,E1 -10626.867,E2 -10626.867} C_VEL
LIN {X 0,Y 411.287,Z 178.752,A -85,B 0,C 180,E1 -10629.838,E2 -10629.838} C_VEL
LIN {X 0,Y 411.299,Z 178.753,A -85,B 0,C 180,E1 -10633.104,E2 -10633.104} C_VEL
LIN {X 0,Y 411.257,Z 178.757,A -85,B 0,C 180,E1 -10636.869,E2 -10636.869} C_VEL
LIN {X 0,Y 411.224,Z 178.757,A -85,B 0,C 180,E1 -10639.986,E2 -10639.986} C_VEL
LIN {X 0,Y 411.197,Z 178.766,A -85,B 0,C 180,E1 -10643.147,E2 -10643.147} C_VEL
LIN {X 0,Y 411.232,Z 178.758,A -85,B 0,C 180,E1 -10646.381,E2 -10646.381} C_VEL
LIN {X 0,Y 411.204,Z 178.76,A -85,B 0,C 180,E1 -10649.712,E2 -10649.712} C_VEL
LIN {X 0,Y 411.2,Z 178.762,A -85,B 0,C 180,E1 -10653.156,E2 -10653.156} C_VEL
LIN {X 0,Y 411.189,Z 178.768,A -85,B 0,C 180,E1 -10656.553,E2 -10656.553} C_VEL
LIN {X 0,Y 411.221,Z 178.758,A -85,B 0,C 180,E1 -10659.73,E2 -10659.73} C_VEL
LIN {X 0,Y 411.171,Z 178.764,A -85,B 0,C 180,E1 -10663.133,E2 -10663.133} C_VEL
LIN {X 0,Y 411.163,Z 178.767,A -85,B 0,C 180,E1 -10665.881,E2 -10665.881} C_VEL
LIN {X 0,Y 411.159,Z 178.767,A -85,B 0,C 180,E1 -10668.772,E2 -10668.772} C_VEL
LIN {X 0,Y 411.206,Z 178.763,A -85,B 0,C 180,E1 -10671.83,E2 -10671.83} C_VEL
LIN {X 0,Y 411.206,Z 178.76,A -85,B 0,C 180,E1 -10675.121,E2 -10675.121} C_VEL
LIN {X 0,Y 411.167,Z 178.771,A -85,B 0,C 180,E1 -10678.003,E2 -10678.003} C_VEL
LIN {X 0,Y 411.219,Z 178.76,A -85,B 0,C 180,E1 -10681.411,E2 -10681.411} C_VEL
LIN {X 0,Y 411.232,Z 178.756,A -85,B 0,C 180,E1 -10684.707,E2 -10684.707} C_VEL
LIN {X 0,Y 411.201,Z 178.764,A -85,B 0,C 180,E1 -10687.914,E2 -10687.914} C_VEL
LIN {X 0,Y 411.22,Z 178.759,A -85,B 0,C 180,E1 -10691.052,E2 -10691.052} C_VEL
LIN {X 0,Y 411.251,Z 178.759,A -85,B 0,C 180,E1 -10694.132,E2 -10694.132} C_VEL
LIN {X 0,Y 411.299,Z 178.754,A -85,B 0,C 180,E1 -10697.166,E2 -10697.166} C_VEL
LIN {X 0,Y 411.29,Z 178.754,A -85,B 0,C 180,E1 -10700.161,E2 -10700.161} C_VEL
LIN {X 0,Y 411.458,Z 178.733,A -85,B 0,C 180,E1 -10703.133,E2 -10703.133} C_VEL
LIN {X 0,Y 411.309,Z 178.753,A -85,B 0,C 180,E1 -10705.099,E2 -10705.099} C_VEL
LIN {X 0,Y 411.511,Z 178.725,A -85,B 0,C 180,E1 -10708.043,E2 -10708.043} C_VEL
LIN {X 0,Y 411.639,Z 178.711,A -85,B 0,C 180,E1 -10710,E2 -10710} C_VEL
LIN {X 0,Y 411.463,Z 178.733,A -85,B 0,C 180,E1 -10712.937,E2 -10712.937} C_VEL
LIN {X 0,Y 411.458,Z 178.733,A -85,B 0,C 180,E1 -10716.867,E2 -10716.867} C_VEL
LIN {X 0,Y 411.29,Z 178.754,A -85,B 0,C 180,E1 -10719.839,E2 -10719.839} C_VEL
LIN {X 0,Y 411.28,Z 178.755,A -85,B 0,C 180,E1 -10723.318,E2 -10723.318} C_VEL
LIN {X 0,Y 411.253,Z 178.759,A -85,B 0,C 180,E1 -10726.889,E2 -10726.889} C_VEL
LIN {X 0,Y 411.236,Z 178.759,A -85,B 0,C 180,E1 -10727.584,E2 -10727.584} C_VEL
LIN {X 0,Y 410.575,Z 178.845,A -85,B 0,C 180,E1 -10728.402,E2 -10728.402} C_VEL
LIN {X 0,Y 407.688,Z 179.2,A -85,B 0,C 180,E1 -10729.73,E2 -10729.73} C_VEL
LIN {X 0,Y 405.244,Z 179.505,A -85,B 0,C 180,E1 -10730.803,E2 -10730.803} C_VEL
LIN {X 0,Y 404.208,Z 179.632,A -85,B 0,C 180,E1 -10731.634,E2 -10731.634} C_VEL
LIN {X 0,Y 404.132,Z 179.641,A -85,B 0,C 180,E1 -10731.915,E2 -10731.915} C_VEL
LIN {X 0,Y 404.211,Z 179.631,A -85,B 0,C 180,E1 -10735.296,E2 -10735.296} C_VEL
LIN {X 0,Y 404.193,Z 179.638,A -85,B 0,C 180,E1 -10737.999,E2 -10737.999} C_VEL
LIN {X 0,Y 404.141,Z 179.641,A -85,B 0,C 180,E1 -10741.56,E2 -10741.56} C_VEL
LIN {X 0,Y 404.18,Z 179.635,A -85,B 0,C 180,E1 -10745.016,E2 -10745.016} C_VEL
LIN {X 0,Y 404.157,Z 179.638,A -85,B 0,C 180,E1 -10748.756,E2 -10748.756} C_VEL
LIN {X 0,Y 404.144,Z 179.644,A -85,B 0,C 180,E1 -10751.604,E2 -10751.604} C_VEL
LIN {X 0,Y 404.14,Z 179.64,A -85,B 0,C 180,E1 -10754.522,E2 -10754.522} C_VEL
LIN {X 0,Y 404.165,Z 179.64,A -85,B 0,C 180,E1 -10757.3,E2 -10757.3} C_VEL
LIN {X 0,Y 404.163,Z 179.639,A -85,B 0,C 180,E1 -10759.955,E2 -10759.955} C_VEL
LIN {X 0,Y 404.134,Z 179.644,A -85,B 0,C 180,E1 -10763.124,E2 -10763.124} C_VEL
LIN {X 0,Y 404.139,Z 179.64,A -85,B 0,C 180,E1 -10766.188,E2 -10766.188} C_VEL
LIN {X 0,Y 404.148,Z 179.641,A -85,B 0,C 180,E1 -10769.716,E2 -10769.716} C_VEL
LIN {X 0,Y 404.19,Z 179.641,A -85,B 0,C 180,E1 -10773.123,E2 -10773.123} C_VEL
LIN {X 0,Y 404.171,Z 179.64,A -85,B 0,C 180,E1 -10775.335,E2 -10775.335} C_VEL
LIN {X 0,Y 404.132,Z 179.644,A -85,B 0,C 180,E1 -10778.581,E2 -10778.581} C_VEL
LIN {X 0,Y 404.204,Z 179.632,A -85,B 0,C 180,E1 -10781.762,E2 -10781.762} C_VEL
LIN {X 0,Y 404.2,Z 179.638,A -85,B 0,C 180,E1 -10784.882,E2 -10784.882} C_VEL
LIN {X 0,Y 404.25,Z 179.627,A -85,B 0,C 180,E1 -10787.959,E2 -10787.959} C_VEL
LIN {X 0,Y 404.399,Z 179.61,A -85,B 0,C 180,E1 -10792.129,E2 -10792.129} C_VEL
LIN {X 0,Y 404.417,Z 179.607,A -85,B 0,C 180,E1 -10794.016,E2 -10794.016} C_VEL
LIN {X 0,Y 404.474,Z 179.601,A -85,B 0,C 180,E1 -10798.009,E2 -10798.009} C_VEL
LIN {X 0,Y 404.605,Z 179.585,A -85,B 0,C 180,E1 -10800.001,E2 -10800.001} C_VEL
LIN {X 0,Y 404.41,Z 179.607,A -85,B 0,C 180,E1 -10802.989,E2 -10802.989} C_VEL
LIN {X 0,Y 404.414,Z 179.611,A -85,B 0,C 180,E1 -10805.986,E2 -10805.986} C_VEL
LIN {X 0,Y 404.286,Z 179.622,A -85,B 0,C 180,E1 -10809.002,E2 -10809.002} C_VEL
LIN {X 0,Y 404.251,Z 179.632,A -85,B 0,C 180,E1 -10812.042,E2 -10812.042} C_VEL
LIN {X 0,Y 404.201,Z 179.633,A -85,B 0,C 180,E1 -10815.119,E2 -10815.119} C_VEL
LIN {X 0,Y 404.206,Z 179.634,A -85,B 0,C 180,E1 -10818.239,E2 -10818.239} C_VEL
LIN {X 0,Y 404.135,Z 179.644,A -85,B 0,C 180,E1 -10821.42,E2 -10821.42} C_VEL
LIN {X 0,Y 404.174,Z 179.636,A -85,B 0,C 180,E1 -10824.666,E2 -10824.666} C_VEL
LIN {X 0,Y 404.192,Z 179.635,A -85,B 0,C 180,E1 -10828,E2 -10828} C_VEL
LIN {X 0,Y 404.137,Z 179.645,A -85,B 0,C 180,E1 -10831.559,E2 -10831.559} C_VEL
LIN {X 0,Y 404.182,Z 179.641,A -85,B 0,C 180,E1 -10835.017,E2 -10835.017} C_VEL
LIN {X 0,Y 404.149,Z 179.645,A -85,B 0,C 180,E1 -10838.758,E2 -10838.758} C_VEL
LIN {X 0,Y 404.286,Z 180.427,A -85,B 0,C 180,E1 -10840.104,E2 -10840.104} C_VEL
LIN {X 0,Y 404.728,Z 183.372,A -85,B 0,C 180,E1 -10843.172,E2 -10843.172} C_VEL
LIN {X 0,Y 405.137,Z 186.389,A -85,B 0,C 180,E1 -10846.062,E2 -10846.062} C_VEL
LIN {X 0,Y 405.317,Z 189.5,A -85,B 0,C 180,E1 -10848.785,E2 -10848.785} C_VEL
LIN {X 0,Y 405.079,Z 192.639,A -85,B 0,C 180,E1 -10851.349,E2 -10851.349} C_VEL
LIN {X 0,Y 404.604,Z 197.479,A -85,B 0,C 180,E1 -10855.026,E2 -10855.026} C_VEL
LIN {X 0,Y 404.196,Z 202.422,A -85,B 0,C 180,E1 -10858.559,E2 -10858.559} C_VEL
LIN {X 0,Y 403.848,Z 207.453,A -85,B 0,C 180,E1 -10861.975,E2 -10861.975} C_VEL
LIN {X 0,Y 403.54,Z 212.556,A -85,B 0,C 180,E1 -10865.293,E2 -10865.293} C_VEL
LIN {X 0,Y 403.307,Z 217.715,A -85,B 0,C 180,E1 -10868.535,E2 -10868.535} C_VEL
LIN {X 0,Y 403.081,Z 222.926,A -85,B 0,C 180,E1 -10871.709,E2 -10871.709} C_VEL
LIN {X 0,Y 403.093,Z 223.653,A -85,B 0,C 180,E1 -10872.122,E2 -10872.122} C_VEL
LIN {X 0,Y 405.057,Z 233.86,A -85,B 0,C 180,E1 -10872.525,E2 -10872.525} C_VEL
LIN {X 0,Y 406.825,Z 243.864,A -85,B 0,C 180,E1 -10873.035,E2 -10873.035} C_VEL
LIN {X 0,Y 407.944,Z 252.66,A -85,B 0,C 180,E1 -10873.573,E2 -10873.573} C_VEL
LIN {X 0,Y 407.334,Z 262.448,A -85,B 0,C 180,E1 -10874.232,E2 -10874.232} C_VEL
LIN {X 0,Y 406.704,Z 271.447,A -85,B 0,C 180,E1 -10874.977,E2 -10874.977} C_VEL
LIN {X 0,Y 406.064,Z 280.03,A -85,B 0,C 180,E1 -10875.833,E2 -10875.833} C_VEL
LIN {X 0,Y 405.546,Z 287.58,A -85,B 0,C 180,E1 -10876.726,E2 -10876.726} C_VEL
LIN {X 0,Y 404.942,Z 294.802,A -85,B 0,C 180,E1 -10877.725,E2 -10877.725} C_VEL
LIN {X 0,Y 404.423,Z 301.007,A -85,B 0,C 180,E1 -10878.726,E2 -10878.726} C_VEL
LIN {X 0,Y 403.922,Z 307.547,A -85,B 0,C 180,E1 -10879.98,E2 -10879.98} C_VEL
LIN {X 0,Y 403.598,Z 312.051,A -85,B 0,C 180,E1 -10880.984,E2 -10880.984} C_VEL
LIN {X 0,Y 403.213,Z 317.544,A -85,B 0,C 180,E1 -10882.489,E2 -10882.489} C_VEL
LIN {X 0,Y 402.996,Z 321.87,A -85,B 0,C 180,E1 -10883.994,E2 -10883.994} C_VEL
LIN {X 0,Y 402.972,Z 324.239,A -85,B 0,C 180,E1 -10884.997,E2 -10884.997} C_VEL
LIN {X 0,Y 402.867,Z 326.036,A -85,B 0,C 180,E1 -10885.999,E2 -10885.999} C_VEL
LIN {X 0,Y 402.862,Z 328.482,A -85,B 0,C 180,E1 -10888.001,E2 -10888.001} C_VEL
LIN {X 0,Y 402.847,Z 329.07,A -85,B 0,C 180,E1 -10889,E2 -10889} C_VEL
LIN {X 0,Y 402.847,Z 329.07,A -85,B 0,C 180,E1 -10891,E2 -10891} C_VEL
LIN {X 0,Y 402.862,Z 328.482,A -85,B 0,C 180,E1 -10891.999,E2 -10891.999} C_VEL
LIN {X 0,Y 402.867,Z 326.036,A -85,B 0,C 180,E1 -10894.001,E2 -10894.001} C_VEL
LIN {X 0,Y 402.966,Z 323.087,A -85,B 0,C 180,E1 -10895.504,E2 -10895.504} C_VEL
LIN {X 0,Y 403.119,Z 319.098,A -85,B 0,C 180,E1 -10897.01,E2 -10897.01} C_VEL
LIN {X 0,Y 403.435,Z 313.967,A -85,B 0,C 180,E1 -10898.515,E2 -10898.515} C_VEL
LIN {X 0,Y 403.842,Z 308.704,A -85,B 0,C 180,E1 -10899.769,E2 -10899.769} C_VEL
LIN {X 0,Y 404.272,Z 302.382,A -85,B 0,C 180,E1 -10901.024,E2 -10901.024} C_VEL
LIN {X 0,Y 404.791,Z 296.43,A -85,B 0,C 180,E1 -10902.025,E2 -10902.025} C_VEL
LIN {X 0,Y 405.37,Z 289.5,A -85,B 0,C 180,E1 -10903.025,E2 -10903.025} C_VEL
LIN {X 0,Y 406.036,Z 281.317,A -85,B 0,C 180,E1 -10904.023,E2 -10904.023} C_VEL
LIN {X 0,Y 406.56,Z 272.764,A -85,B 0,C 180,E1 -10904.903,E2 -10904.903} C_VEL
LIN {X 0,Y 407.217,Z 264.08,A -85,B 0,C 180,E1 -10905.644,E2 -10905.644} C_VEL
LIN {X 0,Y 407.927,Z 254.337,A -85,B 0,C 180,E1 -10906.321,E2 -10906.321} C_VEL
LIN {X 0,Y 407.599,Z 249.278,A -85,B 0,C 180,E1 -10906.656,E2 -10906.656} C_VEL
LIN {X 0,Y 405.482,Z 236.077,A -85,B 0,C 180,E1 -10907.375,E2 -10907.375} C_VEL
LIN {X 0,Y 403.245,Z 224.907,A -85,B 0,C 180,E1 -10907.839,E2 -10907.839} C_VEL
LIN {X 0,Y 403.086,Z 223.627,A -85,B 0,C 180,E1 -10907.893,E2 -10907.893} C_VEL
LIN {X 0,Y 403.24,Z 219.438,A -85,B 0,C 180,E1 -10910.4,E2 -10910.4} C_VEL
LIN {X 0,Y 403.433,Z 214.259,A -85,B 0,C 180,E1 -10913.62,E2 -10913.62} C_VEL
LIN {X 0,Y 403.739,Z 209.137,A -85,B 0,C 180,E1 -10916.909,E2 -10916.909} C_VEL
LIN {X 0,Y 404.048,Z 204.084,A -85,B 0,C 180,E1 -10920.293,E2 -10920.293} C_VEL
LIN {X 0,Y 404.436,Z 199.127,A -85,B 0,C 180,E1 -10923.784,E2 -10923.784} C_VEL
LIN {X 0,Y 404.859,Z 194.772,A -85,B 0,C 180,E1 -10927.01,E2 -10927.01} C_VEL
LIN {X 0,Y 405.228,Z 191.069,A -85,B 0,C 180,E1 -10929.918,E2 -10929.918} C_VEL
LIN {X 0,Y 405.296,Z 187.933,A -85,B 0,C 180,E1 -10932.553,E2 -10932.553} C_VEL
LIN {X 0,Y 404.921,Z 184.86,A -85,B 0,C 180,E1 -10935.366,E2 -10935.366} C_VEL
LIN {X 0,Y 404.444,Z 181.588,A -85,B 0,C 180,E1 -10938.675,E2 -10938.675} C_VEL
LIN {X 0,Y 404.266,Z 180.374,A -85,B 0,C 180,E1 -10939.966,E2 -10939.966} C_VEL
LIN {X 0,Y 404.149,Z 179.644,A -85,B 0,C 180,E1 -10941.492,E2 -10941.492} C_VEL
LIN {X 0,Y 404.182,Z 179.64,A -85,B 0,C 180,E1 -10944.983,E2 -10944.983} C_VEL
LIN {X 0,Y 404.139,Z 179.646,A -85,B 0,C 180,E1 -10948.553,E2 -10948.553} C_VEL
LIN {X 0,Y 404.192,Z 179.635,A -85,B 0,C 180,E1 -10952,E2 -10952} C_VEL
LIN {X 0,Y 404.174,Z 179.636,A -85,B 0,C 180,E1 -10955.334,E2 -10955.334} C_VEL
LIN {X 0,Y 404.135,Z 179.644,A -85,B 0,C 180,E1 -10958.58,E2 -10958.58} C_VEL
LIN {X 0,Y 404.206,Z 179.634,A -85,B 0,C 180,E1 -10961.761,E2 -10961.761} C_VEL
LIN {X 0,Y 404.201,Z 179.633,A -85,B 0,C 180,E1 -10964.881,E2 -10964.881} C_VEL
LIN {X 0,Y 404.251,Z 179.632,A -85,B 0,C 180,E1 -10967.958,E2 -10967.958} C_VEL
LIN {X 0,Y 404.4,Z 179.612,A -85,B 0,C 180,E1 -10972.128,E2 -10972.128} C_VEL
LIN {X 0,Y 404.414,Z 179.611,A -85,B 0,C 180,E1 -10974.014,E2 -10974.014} C_VEL
LIN {X 0,Y 404.474,Z 179.602,A -85,B 0,C 180,E1 -10978.008,E2 -10978.008} C_VEL
LIN {X 0,Y 404.605,Z 179.585,A -85,B 0,C 180,E1 -10979.999,E2 -10979.999} C_VEL
LIN {X 0,Y 404.41,Z 179.607,A -85,B 0,C 180,E1 -10982.988,E2 -10982.988} C_VEL
LIN {X 0,Y 404.39,Z 179.609,A -85,B 0,C 180,E1 -10986.649,E2 -10986.649} C_VEL
LIN {X 0,Y 404.285,Z 179.624,A -85,B 0,C 180,E1 -10989.001,E2 -10989.001} C_VEL
LIN {X 0,Y 404.25,Z 179.627,A -85,B 0,C 180,E1 -10992.041,E2 -10992.041} C_VEL
LIN {X 0,Y 404.2,Z 179.638,A -85,B 0,C 180,E1 -10995.118,E2 -10995.118} C_VEL
LIN {X 0,Y 404.204,Z 179.632,A -85,B 0,C 180,E1 -10998.238,E2 -10998.238} C_VEL
LIN {X 0,Y 404.132,Z 179.644,A -85,B 0,C 180,E1 -11001.419,E2 -11001.419} C_VEL
LIN {X 0,Y 404.171,Z 179.64,A -85,B 0,C 180,E1 -11004.665,E2 -11004.665} C_VEL
LIN {X 0,Y 404.192,Z 179.633,A -85,B 0,C 180,E1 -11007.999,E2 -11007.999} C_VEL
LIN {X 0,Y 404.136,Z 179.64,A -85,B 0,C 180,E1 -11011.559,E2 -11011.559} C_VEL
LIN {X 0,Y 404.179,Z 179.638,A -85,B 0,C 180,E1 -11015.016,E2 -11015.016} C_VEL
LIN {X 0,Y 404.157,Z 179.642,A -85,B 0,C 180,E1 -11018.756,E2 -11018.756} C_VEL
LIN {X 0,Y 404.143,Z 179.639,A -85,B 0,C 180,E1 -11021.604,E2 -11021.604} C_VEL
LIN {X 0,Y 404.139,Z 179.645,A -85,B 0,C 180,E1 -11024.522,E2 -11024.522} C_VEL
LIN {X 0,Y 404.132,Z 179.641,A -85,B 0,C 180,E1 -11027.296,E2 -11027.296} C_VEL
LIN {X 0,Y 404.163,Z 179.641,A -85,B 0,C 180,E1 -11029.955,E2 -11029.955} C_VEL
LIN {X 0,Y 404.134,Z 179.64,A -85,B 0,C 180,E1 -11033.124,E2 -11033.124} C_VEL
LIN {X 0,Y 404.14,Z 179.645,A -85,B 0,C 180,E1 -11036.188,E2 -11036.188} C_VEL
LIN {X 0,Y 404.15,Z 179.643,A -85,B 0,C 180,E1 -11039.716,E2 -11039.716} C_VEL
LIN {X 0,Y 404.191,Z 179.634,A -85,B 0,C 180,E1 -11043.123,E2 -11043.123} C_VEL
LIN {X 0,Y 404.173,Z 179.638,A -85,B 0,C 180,E1 -11045.335,E2 -11045.335} C_VEL
LIN {X 0,Y 404.135,Z 179.64,A -85,B 0,C 180,E1 -11048.581,E2 -11048.581} C_VEL
LIN {X 0,Y 404.206,Z 179.637,A -85,B 0,C 180,E1 -11051.762,E2 -11051.762} C_VEL
LIN {X 0,Y 404.203,Z 179.638,A -85,B 0,C 180,E1 -11054.882,E2 -11054.882} C_VEL
LIN {X 0,Y 404.253,Z 179.629,A -85,B 0,C 180,E1 -11057.959,E2 -11057.959} C_VEL
LIN {X 0,Y 404.43,Z 179.608,A -85,B 0,C 180,E1 -11062.1,E2 -11062.1} C_VEL
LIN {X 0,Y 404.421,Z 179.609,A -85,B 0,C 180,E1 -11064.015,E2 -11064.015} C_VEL
LIN {X 0,Y 404.479,Z 179.601,A -85,B 0,C 180,E1 -11068.009,E2 -11068.009} C_VEL
LIN {X 0,Y 404.608,Z 179.587,A -85,B 0,C 180,E1 -11070,E2 -11070} C_VEL
LIN {X 0,Y 404.42,Z 179.61,A -85,B 0,C 180,E1 -11072.988,E2 -11072.988} C_VEL
LIN {X 0,Y 404.409,Z 179.611,A -85,B 0,C 180,E1 -11076.987,E2 -11076.987} C_VEL
LIN {X 0,Y 404.255,Z 179.631,A -85,B 0,C 180,E1 -11080.012,E2 -11080.012} C_VEL
LIN {X 0,Y 404.262,Z 179.63,A -85,B 0,C 180,E1 -11083.211,E2 -11083.211} C_VEL
LIN {X 0,Y 404.212,Z 179.636,A -85,B 0,C 180,E1 -11087.007,E2 -11087.007} C_VEL
LIN {X 0,Y 404.183,Z 179.641,A -85,B 0,C 180,E1 -11090.35,E2 -11090.35} C_VEL
LIN {X 0,Y 404.132,Z 179.641,A -85,B 0,C 180,E1 -11091.915,E2 -11091.915} C_VEL
LIN {X 0,Y 403.489,Z 179.727,A -85,B 0,C 180,E1 -11092.746,E2 -11092.746} C_VEL
LIN {X 0,Y 400.657,Z 180.087,A -85,B 0,C 180,E1 -11094.098,E2 -11094.098} C_VEL
LIN {X 0,Y 398.247,Z 180.388,A -85,B 0,C 180,E1 -11095.19,E2 -11095.19} C_VEL
LIN {X 0,Y 397.213,Z 180.512,A -85,B 0,C 180,E1 -11096.035,E2 -11096.035} C_VEL
LIN {X 0,Y 397.13,Z 180.519,A -85,B 0,C 180,E1 -11096.32,E2 -11096.32} C_VEL
LIN {X 0,Y 397.122,Z 180.517,A -85,B 0,C 180,E1 -11098.543,E2 -11098.543} C_VEL
LIN {X 0,Y 397.106,Z 180.523,A -85,B 0,C 180,E1 -11102.068,E2 -11102.068} C_VEL
LIN {X 0,Y 397.115,Z 180.517,A -85,B 0,C 180,E1 -11105.504,E2 -11105.504} C_VEL
LIN {X 0,Y 397.131,Z 180.513,A -85,B 0,C 180,E1 -11108.863,E2 -11108.863} C_VEL
LIN {X 0,Y 397.109,Z 180.517,A -85,B 0,C 180,E1 -11112.261,E2 -11112.261} C_VEL
LIN {X 0,Y 397.081,Z 180.52,A -85,B 0,C 180,E1 -11115.069,E2 -11115.069} C_VEL
LIN {X 0,Y 397.104,Z 180.518,A -85,B 0,C 180,E1 -11118.014,E2 -11118.014} C_VEL
LIN {X 0,Y 397.131,Z 180.516,A -85,B 0,C 180,E1 -11121.137,E2 -11121.137} C_VEL
LIN {X 0,Y 397.114,Z 180.515,A -85,B 0,C 180,E1 -11124.497,E2 -11124.497} C_VEL
LIN {X 0,Y 397.074,Z 180.521,A -85,B 0,C 180,E1 -11127.929,E2 -11127.929} C_VEL
LIN {X 0,Y 397.121,Z 180.518,A -85,B 0,C 180,E1 -11131.457,E2 -11131.457} C_VEL
LIN {X 0,Y 397.146,Z 180.512,A -85,B 0,C 180,E1 -11134.488,E2 -11134.488} C_VEL
LIN {X 0,Y 397.103,Z 180.522,A -85,B 0,C 180,E1 -11137.086,E2 -11137.086} C_VEL
LIN {X 0,Y 397.142,Z 180.513,A -85,B 0,C 180,E1 -11140.353,E2 -11140.353} C_VEL
LIN {X 0,Y 397.16,Z 180.51,A -85,B 0,C 180,E1 -11143.554,E2 -11143.554} C_VEL
LIN {X 0,Y 397.223,Z 180.508,A -85,B 0,C 180,E1 -11146.703,E2 -11146.703} C_VEL
LIN {X 0,Y 397.212,Z 180.503,A -85,B 0,C 180,E1 -11149.809,E2 -11149.809} C_VEL
LIN {X 0,Y 397.347,Z 180.489,A -85,B 0,C 180,E1 -11152.888,E2 -11152.888} C_VEL
LIN {X 0,Y 397.248,Z 180.5,A -85,B 0,C 180,E1 -11154.926,E2 -11154.926} C_VEL
LIN {X 0,Y 397.443,Z 180.477,A -85,B 0,C 180,E1 -11157.974,E2 -11157.974} C_VEL
LIN {X 0,Y 397.575,Z 180.461,A -85,B 0,C 180,E1 -11160.001,E2 -11160.001} C_VEL
LIN {X 0,Y 397.369,Z 180.483,A -85,B 0,C 180,E1 -11163.042,E2 -11163.042} C_VEL
LIN {X 0,Y 397.365,Z 180.49,A -85,B 0,C 180,E1 -11166.092,E2 -11166.092} C_VEL
LIN {X 0,Y 397.248,Z 180.498,A -85,B 0,C 180,E1 -11169.162,E2 -11169.162} C_VEL
LIN {X 0,Y 397.215,Z 180.506,A -85,B 0,C 180,E1 -11172.259,E2 -11172.259} C_VEL
LIN {X 0,Y 397.175,Z 180.51,A -85,B 0,C 180,E1 -11175.393,E2 -11175.393} C_VEL
LIN {X 0,Y 397.158,Z 180.51,A -85,B 0,C 180,E1 -11178.574,E2 -11178.574} C_VEL
LIN {X 0,Y 397.093,Z 180.523,A -85,B 0,C 180,E1 -11181.819,E2 -11181.819} C_VEL
LIN {X 0,Y 397.153,Z 180.512,A -85,B 0,C 180,E1 -11185.132,E2 -11185.132} C_VEL
LIN {X 0,Y 397.159,Z 180.513,A -85,B 0,C 180,E1 -11187.777,E2 -11187.777} C_VEL
LIN {X 0,Y 397.076,Z 180.521,A -85,B 0,C 180,E1 -11190.883,E2 -11190.883} C_VEL
LIN {X 0,Y 397.123,Z 180.518,A -85,B 0,C 180,E1 -11194.494,E2 -11194.494} C_VEL
LIN {X 0,Y 397.098,Z 180.524,A -85,B 0,C 180,E1 -11198.276,E2 -11198.276} C_VEL
LIN {X 0,Y 397.11,Z 180.522,A -85,B 0,C 180,E1 -11198.859,E2 -11198.859} C_VEL
LIN {X 0,Y 397.579,Z 183.579,A -85,B 0,C 180,E1 -11202.201,E2 -11202.201} C_VEL
LIN {X 0,Y 397.975,Z 186.434,A -85,B 0,C 180,E1 -11205.06,E2 -11205.06} C_VEL
LIN {X 0,Y 398.316,Z 189.509,A -85,B 0,C 180,E1 -11207.896,E2 -11207.896} C_VEL
LIN {X 0,Y 398.062,Z 193.164,A -85,B 0,C 180,E1 -11210.973,E2 -11210.973} C_VEL
LIN {X 0,Y 397.631,Z 197.538,A -85,B 0,C 180,E1 -11214.394,E2 -11214.394} C_VEL
LIN {X 0,Y 397.164,Z 202.64,A -85,B 0,C 180,E1 -11218.145,E2 -11218.145} C_VEL
LIN {X 0,Y 396.829,Z 207.352,A -85,B 0,C 180,E1 -11221.434,E2 -11221.434} C_VEL
LIN {X 0,Y 396.497,Z 212.425,A -85,B 0,C 180,E1 -11224.824,E2 -11224.824} C_VEL
LIN {X 0,Y 396.269,Z 217.556,A -85,B 0,C 180,E1 -11228.134,E2 -11228.134} C_VEL
LIN {X 0,Y 396.016,Z 222.74,A -85,B 0,C 180,E1 -11231.371,E2 -11231.371} C_VEL
LIN {X 0,Y 396,Z 223.47,A -85,B 0,C 180,E1 -11231.792,E2 -11231.792} C_VEL
LIN {X 0,Y 398.071,Z 233.977,A -85,B 0,C 180,E1 -11232.221,E2 -11232.221} C_VEL
LIN {X 0,Y 399.883,Z 244.108,A -85,B 0,C 180,E1 -11232.755,E2 -11232.755} C_VEL
LIN {X 0,Y 401.033,Z 252.846,A -85,B 0,C 180,E1 -11233.307,E2 -11233.307} C_VEL
LIN {X 0,Y 400.618,Z 260.604,A -85,B 0,C 180,E1 -11233.83,E2 -11233.83} C_VEL
LIN {X 0,Y 399.926,Z 269.883,A -85,B 0,C 180,E1 -11234.586,E2 -11234.586} C_VEL
LIN {X 0,Y 399.206,Z 279.347,A -85,B 0,C 180,E1 -11235.53,E2 -11235.53} C_VEL
LIN {X 0,Y 398.601,Z 287.368,A -85,B 0,C 180,E1 -11236.49,E2 -11236.49} C_VEL
LIN {X 0,Y 397.974,Z 294.59,A -85,B 0,C 180,E1 -11237.507,E2 -11237.507} C_VEL
LIN {X 0,Y 397.43,Z 300.794,A -85,B 0,C 180,E1 -11238.525,E2 -11238.525} C_VEL
LIN {X 0,Y 396.915,Z 307.336,A -85,B 0,C 180,E1 -11239.801,E2 -11239.801} C_VEL
LIN {X 0,Y 396.559,Z 311.839,A -85,B 0,C 180,E1 -11240.822,E2 -11240.822} C_VEL
LIN {X 0,Y 396.163,Z 317.332,A -85,B 0,C 180,E1 -11242.354,E2 -11242.354} C_VEL
LIN {X 0,Y 395.931,Z 321.658,A -85,B 0,C 180,E1 -11243.886,E2 -11243.886} C_VEL
LIN {X 0,Y 395.885,Z 324.027,A -85,B 0,C 180,E1 -11244.908,E2 -11244.908} C_VEL
LIN {X 0,Y 395.791,Z 325.825,A -85,B 0,C 180,E1 -11245.927,E2 -11245.927} C_VEL
LIN {X 0,Y 395.761,Z 328.27,A -85,B 0,C 180,E1 -11247.965,E2 -11247.965} C_VEL
LIN {X 0,Y 395.777,Z 328.86,A -85,B 0,C 180,E1 -11248.983,E2 -11248.983} C_VEL
LIN {X 0,Y 395.777,Z 328.86,A -85,B 0,C 180,E1 -11251.017,E2 -11251.017} C_VEL
LIN {X 0,Y 395.761,Z 328.27,A -85,B 0,C 180,E1 -11252.035,E2 -11252.035} C_VEL
LIN {X 0,Y 395.791,Z 325.825,A -85,B 0,C 180,E1 -11254.073,E2 -11254.073} C_VEL
LIN {X 0,Y 395.871,Z 322.875,A -85,B 0,C 180,E1 -11255.603,E2 -11255.603} C_VEL
LIN {X 0,Y 396.064,Z 318.886,A -85,B 0,C 180,E1 -11257.135,E2 -11257.135} C_VEL
LIN {X 0,Y 396.391,Z 313.755,A -85,B 0,C 180,E1 -11258.668,E2 -11258.668} C_VEL
LIN {X 0,Y 396.808,Z 308.491,A -85,B 0,C 180,E1 -11259.944,E2 -11259.944} C_VEL
LIN {X 0,Y 397.271,Z 302.17,A -85,B 0,C 180,E1 -11261.221,E2 -11261.221} C_VEL
LIN {X 0,Y 397.821,Z 296.217,A -85,B 0,C 180,E1 -11262.239,E2 -11262.239} C_VEL
LIN {X 0,Y 398.416,Z 289.287,A -85,B 0,C 180,E1 -11263.257,E2 -11263.257} C_VEL
LIN {X 0,Y 399.073,Z 281.103,A -85,B 0,C 180,E1 -11264.273,E2 -11264.273} C_VEL
LIN {X 0,Y 399.681,Z 272.722,A -85,B 0,C 180,E1 -11265.15,E2 -11265.15} C_VEL
LIN {X 0,Y 400.366,Z 263.868,A -85,B 0,C 180,E1 -11265.919,E2 -11265.919} C_VEL
LIN {X 0,Y 401.065,Z 254.416,A -85,B 0,C 180,E1 -11266.589,E2 -11266.589} C_VEL
LIN {X 0,Y 400.079,Z 245.887,A -85,B 0,C 180,E1 -11267.146,E2 -11267.146} C_VEL
LIN {X 0,Y 398.308,Z 235.18,A -85,B 0,C 180,E1 -11267.723,E2 -11267.723} C_VEL
LIN {X 0,Y 396.071,Z 224.263,A -85,B 0,C 180,E1 -11268.184,E2 -11268.184} C_VEL
LIN {X 0,Y 396.02,Z 223.441,A -85,B 0,C 180,E1 -11268.223,E2 -11268.223} C_VEL
LIN {X 0,Y 396.163,Z 219.267,A -85,B 0,C 180,E1 -11270.781,E2 -11270.781} C_VEL
LIN {X 0,Y 396.395,Z 214.105,A -85,B 0,C 180,E1 -11274.065,E2 -11274.065} C_VEL
LIN {X 0,Y 396.759,Z 208.672,A -85,B 0,C 180,E1 -11277.664,E2 -11277.664} C_VEL
LIN {X 0,Y 397.054,Z 204.013,A -85,B 0,C 180,E1 -11280.884,E2 -11280.884} C_VEL
LIN {X 0,Y 397.458,Z 199.069,A -85,B 0,C 180,E1 -11284.46,E2 -11284.46} C_VEL
LIN {X 0,Y 397.868,Z 195.259,A -85,B 0,C 180,E1 -11287.355,E2 -11287.355} C_VEL
LIN {X 0,Y 398.242,Z 191.065,A -85,B 0,C 180,E1 -11290.764,E2 -11290.764} C_VEL
LIN {X 0,Y 398.292,Z 189.432,A -85,B 0,C 180,E1 -11292.174,E2 -11292.174} C_VEL
LIN {X 0,Y 397.952,Z 186.298,A -85,B 0,C 180,E1 -11295.055,E2 -11295.055} C_VEL
LIN {X 0,Y 397.521,Z 183.423,A -85,B 0,C 180,E1 -11297.947,E2 -11297.947} C_VEL
LIN {X 0,Y 397.11,Z 180.521,A -85,B 0,C 180,E1 -11301.141,E2 -11301.141} C_VEL
LIN {X 0,Y 397.117,Z 180.519,A -85,B 0,C 180,E1 -11304.496,E2 -11304.496} C_VEL
LIN {X 0,Y 397.076,Z 180.52,A -85,B 0,C 180,E1 -11307.928,E2 -11307.928} C_VEL
LIN {X 0,Y 397.119,Z 180.514,A -85,B 0,C 180,E1 -11311.456,E2 -11311.456} C_VEL
LIN {X 0,Y 397.15,Z 180.517,A -85,B 0,C 180,E1 -11314.487,E2 -11314.487} C_VEL
LIN {X 0,Y 397.106,Z 180.517,A -85,B 0,C 180,E1 -11317.085,E2 -11317.085} C_VEL
LIN {X 0,Y 397.144,Z 180.517,A -85,B 0,C 180,E1 -11320.352,E2 -11320.352} C_VEL
LIN {X 0,Y 397.162,Z 180.51,A -85,B 0,C 180,E1 -11323.552,E2 -11323.552} C_VEL
LIN {X 0,Y 397.224,Z 180.502,A -85,B 0,C 180,E1 -11326.702,E2 -11326.702} C_VEL
LIN {X 0,Y 397.213,Z 180.507,A -85,B 0,C 180,E1 -11329.808,E2 -11329.808} C_VEL
LIN {X 0,Y 397.344,Z 180.486,A -85,B 0,C 180,E1 -11332.887,E2 -11332.887} C_VEL
LIN {X 0,Y 397.247,Z 180.498,A -85,B 0,C 180,E1 -11334.925,E2 -11334.925} C_VEL
LIN {X 0,Y 397.443,Z 180.478,A -85,B 0,C 180,E1 -11337.973,E2 -11337.973} C_VEL
LIN {X 0,Y 397.575,Z 180.461,A -85,B 0,C 180,E1 -11339.999,E2 -11339.999} C_VEL
LIN {X 0,Y 397.37,Z 180.485,A -85,B 0,C 180,E1 -11343.041,E2 -11343.041} C_VEL
LIN {X 0,Y 397.341,Z 180.487,A -85,B 0,C 180,E1 -11346.647,E2 -11346.647} C_VEL
LIN {X 0,Y 397.247,Z 180.502,A -85,B 0,C 180,E1 -11349.161,E2 -11349.161} C_VEL
LIN {X 0,Y 397.213,Z 180.503,A -85,B 0,C 180,E1 -11352.258,E2 -11352.258} C_VEL
LIN {X 0,Y 397.173,Z 180.513,A -85,B 0,C 180,E1 -11355.392,E2 -11355.392} C_VEL
LIN {X 0,Y 397.156,Z 180.511,A -85,B 0,C 180,E1 -11358.573,E2 -11358.573} C_VEL
LIN {X 0,Y 397.09,Z 180.518,A -85,B 0,C 180,E1 -11361.818,E2 -11361.818} C_VEL
LIN {X 0,Y 397.15,Z 180.515,A -85,B 0,C 180,E1 -11365.131,E2 -11365.131} C_VEL
LIN {X 0,Y 397.157,Z 180.51,A -85,B 0,C 180,E1 -11367.776,E2 -11367.776} C_VEL
LIN {X 0,Y 397.079,Z 180.525,A -85,B 0,C 180,E1 -11370.882,E2 -11370.882} C_VEL
LIN {X 0,Y 397.12,Z 180.519,A -85,B 0,C 180,E1 -11374.493,E2 -11374.493} C_VEL
LIN {X 0,Y 397.104,Z 180.52,A -85,B 0,C 180,E1 -11378.274,E2 -11378.274} C_VEL
LIN {X 0,Y 397.106,Z 180.518,A -85,B 0,C 180,E1 -11380.906,E2 -11380.906} C_VEL
LIN {X 0,Y 397.096,Z 180.518,A -85,B 0,C 180,E1 -11383.648,E2 -11383.648} C_VEL
LIN {X 0,Y 397.097,Z 180.521,A -85,B 0,C 180,E1 -11386.521,E2 -11386.521} C_VEL
LIN {X 0,Y 397.109,Z 180.52,A -85,B 0,C 180,E1 -11390.423,E2 -11390.423} C_VEL
LIN {X 0,Y 397.104,Z 180.521,A -85,B 0,C 180,E1 -11394.266,E2 -11394.266} C_VEL
LIN {X 0,Y 397.11,Z 180.516,A -85,B 0,C 180,E1 -11396.727,E2 -11396.727} C_VEL
LIN {X 0,Y 397.129,Z 180.516,A -85,B 0,C 180,E1 -11400.297,E2 -11400.297} C_VEL
LIN {X 0,Y 397.19,Z 180.506,A -85,B 0,C 180,E1 -11402.61,E2 -11402.61} C_VEL
LIN {X 0,Y 397.129,Z 180.517,A -85,B 0,C 180,E1 -11405.982,E2 -11405.982} C_VEL
LIN {X 0,Y 397.14,Z 180.518,A -85,B 0,C 180,E1 -11409.703,E2 -11409.703} C_VEL
LIN {X 0,Y 397.178,Z 180.512,A -85,B 0,C 180,E1 -11412.845,E2 -11412.845} C_VEL
LIN {X 0,Y 397.223,Z 180.507,A -85,B 0,C 180,E1 -11416.679,E2 -11416.679} C_VEL
LIN {X 0,Y 397.215,Z 180.508,A -85,B 0,C 180,E1 -11419.809,E2 -11419.809} C_VEL
LIN {X 0,Y 397.361,Z 180.489,A -85,B 0,C 180,E1 -11422.888,E2 -11422.888} C_VEL
LIN {X 0,Y 397.253,Z 180.504,A -85,B 0,C 180,E1 -11424.925,E2 -11424.925} C_VEL
LIN {X 0,Y 397.448,Z 180.477,A -85,B 0,C 180,E1 -11427.973,E2 -11427.973} C_VEL
LIN {X 0,Y 397.578,Z 180.463,A -85,B 0,C 180,E1 -11430,E2 -11430} C_VEL
LIN {X 0,Y 397.378,Z 180.486,A -85,B 0,C 180,E1 -11433.041,E2 -11433.041} C_VEL
LIN {X 0,Y 397.361,Z 180.489,A -85,B 0,C 180,E1 -11437.112,E2 -11437.112} C_VEL
LIN {X 0,Y 397.215,Z 180.508,A -85,B 0,C 180,E1 -11440.191,E2 -11440.191} C_VEL
LIN {X 0,Y 397.223,Z 180.507,A -85,B 0,C 180,E1 -11443.321,E2 -11443.321} C_VEL
LIN {X 0,Y 397.178,Z 180.512,A -85,B 0,C 180,E1 -11447.155,E2 -11447.155} C_VEL
LIN {X 0,Y 397.11,Z 180.519,A -85,B 0,C 180,E1 -11450.729,E2 -11450.729} C_VEL
LIN {X 0,Y 397.129,Z 180.517,A -85,B 0,C 180,E1 -11454.018,E2 -11454.018} C_VEL
LIN {X 0,Y 397.13,Z 180.519,A -85,B 0,C 180,E1 -11456.32,E2 -11456.32} C_VEL
LIN {X 0,Y 396.459,Z 180.597,A -85,B 0,C 180,E1 -11457.167,E2 -11457.167} C_VEL
LIN {X 0,Y 393.583,Z 180.957,A -85,B 0,C 180,E1 -11458.543,E2 -11458.543} C_VEL
LIN {X 0,Y 391.149,Z 181.262,A -85,B 0,C 180,E1 -11459.654,E2 -11459.654} C_VEL
LIN {X 0,Y 390.104,Z 181.391,A -85,B 0,C 180,E1 -11460.514,E2 -11460.514} C_VEL
LIN {X 0,Y 390.02,Z 181.399,A -85,B 0,C 180,E1 -11460.806,E2 -11460.806} C_VEL
LIN {X 0,Y 390.063,Z 181.4,A -85,B 0,C 180,E1 -11464.025,E2 -11464.025} C_VEL
LIN {X 0,Y 390.042,Z 181.399,A -85,B 0,C 180,E1 -11467.551,E2 -11467.551} C_VEL
LIN {X 0,Y 390.071,Z 181.392,A -85,B 0,C 180,E1 -11470.825,E2 -11470.825} C_VEL
LIN {X 0,Y 390.05,Z 181.399,A -85,B 0,C 180,E1 -11473.886,E2 -11473.886} C_VEL
LIN {X 0,Y 390.074,Z 181.398,A -85,B 0,C 180,E1 -11477.62,E2 -11477.62} C_VEL
LIN {X 0,Y 390.089,Z 181.391,A -85,B 0,C 180,E1 -11480.908,E2 -11480.908} C_VEL
LIN {X 0,Y 390.079,Z 181.393,A -85,B 0,C 180,E1 -11484.793,E2 -11484.793} C_VEL
LIN {X 0,Y 390.021,Z 181.399,A -85,B 0,C 180,E1 -11488.496,E2 -11488.496} C_VEL
LIN {X 0,Y 390.111,Z 181.387,A -85,B 0,C 180,E1 -11492.07,E2 -11492.07} C_VEL
LIN {X 0,Y 390.074,Z 181.394,A -85,B 0,C 180,E1 -11495.52,E2 -11495.52} C_VEL
LIN {X 0,Y 390.049,Z 181.401,A -85,B 0,C 180,E1 -11498.878,E2 -11498.878} C_VEL
LIN {X 0,Y 390.122,Z 181.387,A -85,B 0,C 180,E1 -11502.167,E2 -11502.167} C_VEL
LIN {X 0,Y 390.138,Z 181.385,A -85,B 0,C 180,E1 -11505.393,E2 -11505.393} C_VEL
LIN {X 0,Y 390.142,Z 181.389,A -85,B 0,C 180,E1 -11508.572,E2 -11508.572} C_VEL
LIN {X 0,Y 390.302,Z 181.365,A -85,B 0,C 180,E1 -11512.032,E2 -11512.032} C_VEL
LIN {X 0,Y 390.22,Z 181.377,A -85,B 0,C 180,E1 -11514.834,E2 -11514.834} C_VEL
LIN {X 0,Y 390.412,Z 181.352,A -85,B 0,C 180,E1 -11517.937,E2 -11517.937} C_VEL
LIN {X 0,Y 390.544,Z 181.337,A -85,B 0,C 180,E1 -11520.001,E2 -11520.001} C_VEL
LIN {X 0,Y 390.304,Z 181.363,A -85,B 0,C 180,E1 -11523.097,E2 -11523.097} C_VEL
LIN {X 0,Y 390.319,Z 181.367,A -85,B 0,C 180,E1 -11526.203,E2 -11526.203} C_VEL
LIN {X 0,Y 390.2,Z 181.377,A -85,B 0,C 180,E1 -11529.329,E2 -11529.329} C_VEL
LIN {X 0,Y 390.19,Z 181.379,A -85,B 0,C 180,E1 -11533.439,E2 -11533.439} C_VEL
LIN {X 0,Y 390.145,Z 181.385,A -85,B 0,C 180,E1 -11537.308,E2 -11537.308} C_VEL
LIN {X 0,Y 390.084,Z 181.391,A -85,B 0,C 180,E1 -11540.471,E2 -11540.471} C_VEL
LIN {X 0,Y 390.086,Z 181.394,A -85,B 0,C 180,E1 -11543.352,E2 -11543.352} C_VEL
LIN {X 0,Y 390.11,Z 181.388,A -85,B 0,C 180,E1 -11546.769,E2 -11546.769} C_VEL
LIN {X 0,Y 390.036,Z 181.397,A -85,B 0,C 180,E1 -11550.301,E2 -11550.301} C_VEL
LIN {X 0,Y 390.066,Z 181.397,A -85,B 0,C 180,E1 -11554.025,E2 -11554.025} C_VEL
LIN {X 0,Y 390.04,Z 181.403,A -85,B 0,C 180,E1 -11557.551,E2 -11557.551} C_VEL
LIN {X 0,Y 390.161,Z 182.033,A -85,B 0,C 180,E1 -11559.236,E2 -11559.236} C_VEL
LIN {X 0,Y 390.592,Z 184.968,A -85,B 0,C 180,E1 -11562.463,E2 -11562.463} C_VEL
LIN {X 0,Y 391.058,Z 188.465,A -85,B 0,C 180,E1 -11565.962,E2 -11565.962} C_VEL
LIN {X 0,Y 391.25,Z 191.054,A -85,B 0,C 180,E1 -11568.347,E2 -11568.347} C_VEL
LIN {X 0,Y 391.017,Z 194.216,A -85,B 0,C 180,E1 -11571.019,E2 -11571.019} C_VEL
LIN {X 0,Y 390.628,Z 197.999,A -85,B 0,C 180,E1 -11574.06,E2 -11574.06} C_VEL
LIN {X 0,Y 390.176,Z 202.278,A -85,B 0,C 180,E1 -11577.292,E2 -11577.292} C_VEL
LIN {X 0,Y 389.817,Z 207.249,A -85,B 0,C 180,E1 -11580.871,E2 -11580.871} C_VEL
LIN {X 0,Y 389.466,Z 212.294,A -85,B 0,C 180,E1 -11584.337,E2 -11584.337} C_VEL
LIN {X 0,Y 389.22,Z 217.396,A -85,B 0,C 180,E1 -11587.717,E2 -11587.717} C_VEL
LIN {X 0,Y 388.98,Z 222.554,A -85,B 0,C 180,E1 -11591.021,E2 -11591.021} C_VEL
LIN {X 0,Y 388.935,Z 223.315,A -85,B 0,C 180,E1 -11591.452,E2 -11591.452} C_VEL
LIN {X 0,Y 391,Z 233.41,A -85,B 0,C 180,E1 -11591.875,E2 -11591.875} C_VEL
LIN {X 0,Y 392.562,Z 242.52,A -85,B 0,C 180,E1 -11592.352,E2 -11592.352} C_VEL
LIN {X 0,Y 393.894,Z 251.498,A -85,B 0,C 180,E1 -11592.921,E2 -11592.921} C_VEL
LIN {X 0,Y 394.13,Z 255.966,A -85,B 0,C 180,E1 -11593.227,E2 -11593.227} C_VEL
LIN {X 0,Y 393.183,Z 268.319,A -85,B 0,C 180,E1 -11594.182,E2 -11594.182} C_VEL
LIN {X 0,Y 392.349,Z 278.625,A -85,B 0,C 180,E1 -11595.212,E2 -11595.212} C_VEL
LIN {X 0,Y 391.634,Z 287.304,A -85,B 0,C 180,E1 -11596.266,E2 -11596.266} C_VEL
LIN {X 0,Y 391.024,Z 294.378,A -85,B 0,C 180,E1 -11597.281,E2 -11597.281} C_VEL
LIN {X 0,Y 390.416,Z 300.581,A -85,B 0,C 180,E1 -11598.316,E2 -11598.316} C_VEL
LIN {X 0,Y 389.896,Z 307.123,A -85,B 0,C 180,E1 -11599.616,E2 -11599.616} C_VEL
LIN {X 0,Y 389.496,Z 311.626,A -85,B 0,C 180,E1 -11600.654,E2 -11600.654} C_VEL
LIN {X 0,Y 389.095,Z 317.12,A -85,B 0,C 180,E1 -11602.214,E2 -11602.214} C_VEL
LIN {X 0,Y 388.856,Z 321.447,A -85,B 0,C 180,E1 -11603.775,E2 -11603.775} C_VEL
LIN {X 0,Y 388.78,Z 323.815,A -85,B 0,C 180,E1 -11604.814,E2 -11604.814} C_VEL
LIN {X 0,Y 388.717,Z 325.614,A -85,B 0,C 180,E1 -11605.853,E2 -11605.853} C_VEL
LIN {X 0,Y 388.659,Z 328.059,A -85,B 0,C 180,E1 -11607.927,E2 -11607.927} C_VEL
LIN {X 0,Y 388.69,Z 328.649,A -85,B 0,C 180,E1 -11608.964,E2 -11608.964} C_VEL
LIN {X 0,Y 388.69,Z 328.649,A -85,B 0,C 180,E1 -11611.036,E2 -11611.036} C_VEL
LIN {X 0,Y 388.659,Z 328.059,A -85,B 0,C 180,E1 -11612.073,E2 -11612.073} C_VEL
LIN {X 0,Y 388.717,Z 325.614,A -85,B 0,C 180,E1 -11614.147,E2 -11614.147} C_VEL
LIN {X 0,Y 388.781,Z 323.815,A -85,B 0,C 180,E1 -11615.186,E2 -11615.186} C_VEL
LIN {X 0,Y 388.917,Z 320.207,A -85,B 0,C 180,E1 -11616.745,E2 -11616.745} C_VEL
LIN {X 0,Y 389.214,Z 315.459,A -85,B 0,C 180,E1 -11618.306,E2 -11618.306} C_VEL
LIN {X 0,Y 389.7,Z 309.435,A -85,B 0,C 180,E1 -11619.865,E2 -11619.865} C_VEL
LIN {X 0,Y 390.155,Z 303.334,A -85,B 0,C 180,E1 -11621.165,E2 -11621.165} C_VEL
LIN {X 0,Y 390.717,Z 297.633,A -85,B 0,C 180,E1 -11622.201,E2 -11622.201} C_VEL
LIN {X 0,Y 391.464,Z 289.075,A -85,B 0,C 180,E1 -11623.497,E2 -11623.497} C_VEL
LIN {X 0,Y 392.147,Z 280.89,A -85,B 0,C 180,E1 -11624.531,E2 -11624.531} C_VEL
LIN {X 0,Y 392.809,Z 272.51,A -85,B 0,C 180,E1 -11625.421,E2 -11625.421} C_VEL
LIN {X 0,Y 393.527,Z 263.656,A -85,B 0,C 180,E1 -11626.203,E2 -11626.203} C_VEL
LIN {X 0,Y 394.202,Z 254.479,A -85,B 0,C 180,E1 -11626.869,E2 -11626.869} C_VEL
LIN {X 0,Y 393.017,Z 245.248,A -85,B 0,C 180,E1 -11627.485,E2 -11627.485} C_VEL
LIN {X 0,Y 391.26,Z 234.854,A -85,B 0,C 180,E1 -11628.057,E2 -11628.057} C_VEL
LIN {X 0,Y 389,Z 224.041,A -85,B 0,C 180,E1 -11628.527,E2 -11628.527} C_VEL
LIN {X 0,Y 388.928,Z 223.255,A -85,B 0,C 180,E1 -11628.568,E2 -11628.568} C_VEL
LIN {X 0,Y 389.121,Z 219.078,A -85,B 0,C 180,E1 -11631.175,E2 -11631.175} C_VEL
LIN {X 0,Y 389.266,Z 215.667,A -85,B 0,C 180,E1 -11633.403,E2 -11633.403} C_VEL
LIN {X 0,Y 389.581,Z 210.602,A -85,B 0,C 180,E1 -11636.807,E2 -11636.807} C_VEL
LIN {X 0,Y 389.934,Z 205.588,A -85,B 0,C 180,E1 -11640.308,E2 -11640.308} C_VEL
LIN {X 0,Y 390.377,Z 200.427,A -85,B 0,C 180,E1 -11644.091,E2 -11644.091} C_VEL
LIN {X 0,Y 390.876,Z 195.78,A -85,B 0,C 180,E1 -11647.708,E2 -11647.708} C_VEL
LIN {X 0,Y 391.175,Z 192.624,A -85,B 0,C 180,E1 -11650.299,E2 -11650.299} C_VEL
LIN {X 0,Y 391.184,Z 189.498,A -85,B 0,C 180,E1 -11653.055,E2 -11653.055} C_VEL
LIN {X 0,Y 390.779,Z 186.448,A -85,B 0,C 180,E1 -11656.003,E2 -11656.003} C_VEL
LIN {X 0,Y 390.33,Z 183.055,A -85,B 0,C 180,E1 -11659.594,E2 -11659.594} C_VEL
LIN {X 0,Y 390.13,Z 181.908,A -85,B 0,C 180,E1 -11660.912,E2 -11660.912} C_VEL
LIN {X 0,Y 390.04,Z 181.402,A -85,B 0,C 180,E1 -11662.449,E2 -11662.449} C_VEL
LIN {X 0,Y 390.066,Z 181.396,A -85,B 0,C 180,E1 -11665.975,E2 -11665.975} C_VEL
LIN {X 0,Y 390.044,Z 181.396,A -85,B 0,C 180,E1 -11669.868,E2 -11669.868} C_VEL
LIN {X 0,Y 390.11,Z 181.388,A -85,B 0,C 180,E1 -11673.231,E2 -11673.231} C_VEL
LIN {X 0,Y 390.103,Z 181.391,A -85,B 0,C 180,E1 -11676.75,E2 -11676.75} C_VEL
LIN {X 0,Y 390.1,Z 181.392,A -85,B 0,C 180,E1 -11679.982,E2 -11679.982} C_VEL
LIN {X 0,Y 390.134,Z 181.385,A -85,B 0,C 180,E1 -11683.247,E2 -11683.247} C_VEL
LIN {X 0,Y 390.19,Z 181.379,A -85,B 0,C 180,E1 -11686.561,E2 -11686.561} C_VEL
LIN {X 0,Y 390.2,Z 181.377,A -85,B 0,C 180,E1 -11690.671,E2 -11690.671} C_VEL
LIN {X 0,Y 390.319,Z 181.367,A -85,B 0,C 180,E1 -11693.797,E2 -11693.797} C_VEL
LIN {X 0,Y 390.412,Z 181.355,A -85,B 0,C 180,E1 -11697.936,E2 -11697.936} C_VEL
LIN {X 0,Y 390.544,Z 181.337,A -85,B 0,C 180,E1 -11699.999,E2 -11699.999} C_VEL
LIN {X 0,Y 390.305,Z 181.365,A -85,B 0,C 180,E1 -11703.096,E2 -11703.096} C_VEL
LIN {X 0,Y 390.296,Z 181.365,A -85,B 0,C 180,E1 -11706.643,E2 -11706.643} C_VEL
LIN {X 0,Y 390.199,Z 181.382,A -85,B 0,C 180,E1 -11709.328,E2 -11709.328} C_VEL
LIN {X 0,Y 390.189,Z 181.383,A -85,B 0,C 180,E1 -11713.438,E2 -11713.438} C_VEL
LIN {X 0,Y 390.143,Z 181.389,A -85,B 0,C 180,E1 -11717.307,E2 -11717.307} C_VEL
LIN {X 0,Y 390.081,Z 181.392,A -85,B 0,C 180,E1 -11720.47,E2 -11720.47} C_VEL
LIN {X 0,Y 390.083,Z 181.394,A -85,B 0,C 180,E1 -11723.351,E2 -11723.351} C_VEL
LIN {X 0,Y 390.108,Z 181.393,A -85,B 0,C 180,E1 -11726.768,E2 -11726.768} C_VEL
LIN {X 0,Y 390.038,Z 181.398,A -85,B 0,C 180,E1 -11730.299,E2 -11730.299} C_VEL
LIN {X 0,Y 390.062,Z 181.394,A -85,B 0,C 180,E1 -11734.024,E2 -11734.024} C_VEL
LIN {X 0,Y 390.041,Z 181.396,A -85,B 0,C 180,E1 -11737.551,E2 -11737.551} C_VEL
LIN {X 0,Y 390.071,Z 181.395,A -85,B 0,C 180,E1 -11740.825,E2 -11740.825} C_VEL
LIN {X 0,Y 390.049,Z 181.397,A -85,B 0,C 180,E1 -11743.886,E2 -11743.886} C_VEL
LIN {X 0,Y 390.052,Z 181.396,A -85,B 0,C 180,E1 -11746.79,E2 -11746.79} C_VEL
LIN {X 0,Y 390.052,Z 181.396,A -85,B 0,C 180,E1 -11749.561,E2 -11749.561} C_VEL
LIN {X 0,Y 390.04,Z 181.399,A -85,B 0,C 180,E1 -11752.449,E2 -11752.449} C_VEL
LIN {X 0,Y 390.079,Z 181.398,A -85,B 0,C 180,E1 -11756.047,E2 -11756.047} C_VEL
LIN {X 0,Y 390.04,Z 181.401,A -85,B 0,C 180,E1 -11759.701,E2 -11759.701} C_VEL
LIN {X 0,Y 390.109,Z 181.389,A -85,B 0,C 180,E1 -11763.232,E2 -11763.232} C_VEL
LIN {X 0,Y 390.102,Z 181.389,A -85,B 0,C 180,E1 -11766.75,E2 -11766.75} C_VEL
LIN {X 0,Y 390.103,Z 181.393,A -85,B 0,C 180,E1 -11769.983,E2 -11769.983} C_VEL
LIN {X 0,Y 390.134,Z 181.39,A -85,B 0,C 180,E1 -11773.248,E2 -11773.248} C_VEL
LIN {X 0,Y 390.19,Z 181.383,A -85,B 0,C 180,E1 -11776.562,E2 -11776.562} C_VEL
LIN {X 0,Y 390.201,Z 181.38,A -85,B 0,C 180,E1 -11780.671,E2 -11780.671} C_VEL
LIN {X 0,Y 390.35,Z 181.571,A -85,B 0,C 180,E1 -11782.704,E2 -11782.704} C_VEL
LIN {X 0,Y 390.911,Z 183.473,A -85,B 0,C 180,E1 -11783.159,E2 -11783.159} C_VEL
LIN {X 0,Y 392.539,Z 185.757,A -85,B 0,C 180,E1 -11784.349,E2 -11784.349} C_VEL
LIN {X 0,Y 394.308,Z 187.018,A -85,B 0,C 180,E1 -11785.912,E2 -11785.912} C_VEL
LIN {X 0,Y 395.197,Z 187.229,A -85,B 0,C 180,E1 -11786.942,E2 -11786.942} C_VEL
LIN {X 0,Y 396.207,Z 187.461,A -85,B 0,C 180,E1 -11788.984,E2 -11788.984} C_VEL
LIN {X 0,Y 396.373,Z 187.46,A -85,B 0,C 180,E1 -11790,E2 -11790} C_VEL
LIN {X 0,Y 395.807,Z 187.384,A -85,B 0,C 180,E1 -11792.035,E2 -11792.035} C_VEL
LIN {X 0,Y 394.474,Z 187.06,A -85,B 0,C 180,E1 -11793.894,E2 -11793.894} C_VEL
LIN {X 0,Y 392.69,Z 185.905,A -85,B 0,C 180,E1 -11795.52,E2 -11795.52} C_VEL
LIN {X 0,Y 390.994,Z 183.649,A -85,B 0,C 180,E1 -11796.774,E2 -11796.774} C_VEL
LIN {X 0,Y 390.385,Z 181.732,A -85,B 0,C 180,E1 -11797.268,E2 -11797.268} C_VEL
LIN {X 0,Y 390.316,Z 181.368,A -85,B 0,C 180,E1 -11797.353,E2 -11797.353} C_VEL
LIN {X 0,Y 390.165,Z 181.385,A -85,B 0,C 180,E1 -11800.377,E2 -11800.377} C_VEL
LIN {X 0,Y 390.166,Z 181.386,A -85,B 0,C 180,E1 -11803.542,E2 -11803.542} C_VEL
LIN {X 0,Y 390.144,Z 181.388,A -85,B 0,C 180,E1 -11807.308,E2 -11807.308} C_VEL
LIN {X 0,Y 390.088,Z 181.396,A -85,B 0,C 180,E1 -11810.472,E2 -11810.472} C_VEL
LIN {X 0,Y 390.085,Z 181.391,A -85,B 0,C 180,E1 -11813.351,E2 -11813.351} C_VEL
LIN {X 0,Y 390.109,Z 181.389,A -85,B 0,C 180,E1 -11816.768,E2 -11816.768} C_VEL
LIN {X 0,Y 390.04,Z 181.401,A -85,B 0,C 180,E1 -11820.299,E2 -11820.299} C_VEL
LIN {X 0,Y 390.02,Z 181.399,A -85,B 0,C 180,E1 -11820.806,E2 -11820.806} C_VEL
LIN {X 0,Y 389.354,Z 181.486,A -85,B 0,C 180,E1 -11821.668,E2 -11821.668} C_VEL
LIN {X 0,Y 386.501,Z 181.837,A -85,B 0,C 180,E1 -11823.069,E2 -11823.069} C_VEL
LIN {X 0,Y 384.094,Z 182.141,A -85,B 0,C 180,E1 -11824.202,E2 -11824.202} C_VEL
LIN {X 0,Y 383.071,Z 182.265,A -85,B 0,C 180,E1 -11825.078,E2 -11825.078} C_VEL
LIN {X 0,Y 382.994,Z 182.275,A -85,B 0,C 180,E1 -11825.374,E2 -11825.374} C_VEL
LIN {X 0,Y 383.003,Z 182.273,A -85,B 0,C 180,E1 -11828.6,E2 -11828.6} C_VEL
LIN {X 0,Y 383.008,Z 182.275,A -85,B 0,C 180,E1 -11831.343,E2 -11831.343} C_VEL
LIN {X 0,Y 382.991,Z 182.275,A -85,B 0,C 180,E1 -11834.303,E2 -11834.303} C_VEL
LIN {X 0,Y 383.033,Z 182.272,A -85,B 0,C 180,E1 -11837.244,E2 -11837.244} C_VEL
LIN {X 0,Y 383.016,Z 182.271,A -85,B 0,C 180,E1 -11840.412,E2 -11840.412} C_VEL
LIN {X 0,Y 383.021,Z 182.271,A -85,B 0,C 180,E1 -11844.045,E2 -11844.045} C_VEL
LIN {X 0,Y 382.982,Z 182.279,A -85,B 0,C 180,E1 -11847.578,E2 -11847.578} C_VEL
